//generate traj
t := count*deltaT;
landVel := -0.05 / period;
decTime := 0.1;
IF isContact(count,legID) = FALSE THEN
	IF t <= allContactTime + period THEN
		objSpline(x:=tp,y:=xp,dy0:=0,dy4:=0,      xt:=t,yt=>tipPos[legID].data[0],vt=>tipVel[legID].data[0]);
		objSpline(x:=tp,y:=yp,dy0:=0,dy4:=0,      xt:=t,yt=>tipPos[legID].data[1],vt=>tipVel[legID].data[1]);
		objSpline(x:=tp,y:=zp,dy0:=0,dy4:=landVel,xt:=t,yt=>tipPos[legID].data[2],vt=>tipVel[legID].data[2]);
	ELSE
		tipPos[legID].data[2] := tipPos[legID].data[2] + landVel*deltaT;//到达目标位置后继续下探
	END_IF
ELSE
	//强制停止，没有减速过程。减速过程的运动距离会导致机器人被顶起来
	FOR i:=0 TO 2 DO
		tipPos[legID].data[i] := tipPos[legID].data[i];
		tipVel[legID].data[i] := 0;
	END_FOR
	(*IF VecNorm(tipVel[legID]) > 1E-3 THEN
		FOR i:=0 TO 2 DO
			acc := -tipVel[legID].data[i] / decTime;
			tipPos[legID].data[i] := tipPos[legID].data[i] + tipVel[legID].data[i]*deltaT + 0.5*acc*deltaT*deltaT;
			tipVel[legID].data[i] := tipVel[legID].data[i] + acc*deltaT;
		END_FOR
	ELSE
		FOR i:=0 TO 2 DO
			tipPos[legID].data[i] := tipPos[legID].data[i];
			tipVel[legID].data[i] := 0;
		END_FOR
	END_IF*)
END_IF
END_METHOD

METHOD UpdateInitAndTrgt : BOOL
VAR_INPUT
END_VAR
VAR
	i: INT;
	bodyDist2T: Vec3;
	tipBias : Vec3;
	rotHalfYaw : Mat3;
END_VAR
//1.确定身体初始和目标位置、速度
//位置速度更新
bodyPosInit := bodyPos;
bodyVelInit := bodyVel;
bodyRPYInit := bodyRPY;
bodyOmgInit := bodyOmg;

//位姿计算：姿态在地面坐标系描述，位置在bodyTrgt坐标系描述
bodyRPYTrgt.data[2] := bodyRPYInit.data[2] + stepYaw;//yaw
CalcSlope(yaw := bodyRPYTrgt.data[2],
		  roll => bodyRPYTrgt.data[0], pitch => bodyRPYTrgt.data[1],
		  deltaH => bodyDist2T.data[2],tipDelta => tipBias);
//bodyRPYTrgt.data[0] := gvl.rpy_model[0] + bodyRPYTrgt.data[0] - bodyRPYInit.data[0];//引入实际角度修正
//bodyRPYTrgt.data[1] := gvl.rpy_model[1] + bodyRPYTrgt.data[1] - bodyRPYInit.data[1];//引入实际角度修正
objRotMtx(yaw:=bodyRPYTrgt.data[2],pitch:=bodyRPYTrgt.data[1],roll:=bodyRPYTrgt.data[0],
		  rm=>bodyPmxTrgt);

Arc2Line(arcLen:=stepL,angle:=stepYaw,lineLen=>stepL);
bodyDist2T.data[0] := stepL*COS(stepDir)*COS(-stepYaw/2)-stepL*SIN(stepDir)*SIN(-stepYaw/2);//身体转yaw时，位置只转yaw/2
bodyDist2T.data[1] := stepL*COS(stepDir)*SIN(-stepYaw/2)+stepL*SIN(stepDir)*COS(-stepYaw/2);

bodyPosTrgt := VecAdd(bodyPosInit,MatMulVec(bodyPmxTrgt,bodyDist2T));
bodyPosInit2T := VecNeg(bodyDist2T);
bodyVelInit2T := MatMulVec(MatTranspose(bodyPmxTrgt),bodyVelInit);

//2.确定摆动腿初始和目标位置，速度总为0
tipPosInit := tipPos;

objRotMtx(yaw:=stepYaw/2,pitch:=0,roll:=0,rm=>rotHalfYaw);
FOR i:=0 TO 5 DO
	tipPosTrgt2T[i] := MatMulVec(rotHalfYaw,VecAdd(tipPosTrgtBase[i],SetVec3(stepL/2*COS(stepDir),stepL/2*SIN(stepDir),0)));
	//tipPosTrgt[i] := VecAdd(VecAdd(MatMulVec(bodyPmxTrgt,tipPosTrgt2T[i]),bodyPosTrgt),tipBias);
	tipPosTrgt[i] := VecAdd(MatMulVec(bodyPmxTrgt,tipPosTrgt2T[i]),bodyPosTrgt);
END_FOR
END_METHOD

METHOD WatchDog : BOOL
VAR_INPUT
	count: UDINT;
END_VAR
IF isFeed=TRUE THEN
	starveCount := count + TRUNC(gvl.sampleRate*0.5);//0.5 second
	isFeed := FALSE;
END_IF

IF count>=starveCount THEN
	cmdL := 0;
	cmdLa := 0;
	cmdYaw := 0;
END_IF
END_METHOD

END_FUNCTION_BLOCK

// ---- POUs/tools/VectorMath/VecNormalize.TcPOU
FUNCTION VecNormalize : Vec3
VAR_INPUT
	a : Vec3;
END_VAR
VAR
END_VAR

VecNormalize := VecMulNum(a, 1/VecNorm(a));

END_FUNCTION

// ---- POUs/tools/VectorMath/VecNorm.TcPOU
FUNCTION VecNorm : lreal
VAR_INPUT
	a : Vec3;
END_VAR
VAR
END_VAR

VecNorm := SQRT(a.data[0] * a.data[0] + a.data[1] * a.data[1] + a.data[2] * a.data[2]);

END_FUNCTION

// ---- POUs/tools/VectorMath/VecCross.TcPOU
FUNCTION VecCross : Vec3
VAR_INPUT
	a, b : Vec3;
END_VAR
VAR
	a1, a2, a3 : LREAL;
	b1, b2, b3 : LREAL;
END_VAR

a1 := a.data[0];
a2 := a.data[1];
a3 := a.data[2];
b1 := b.data[0];
b2 := b.data[1];
b3 := b.data[2];

VecCross.data[0] := a2*b3 - a3*b2;
VecCross.data[1] := a3*b1 - a1*b3;
VecCross.data[2] := a1*b2 - a2*b1;

END_FUNCTION

// ---- POUs/tools/VectorMath/Atan2.TcPOU
FUNCTION Atan2 : LREAL//输出角度范围为[-pi,pi]
VAR_INPUT
	y : LREAL;
	x : LREAL;
END_VAR
VAR
END_VAR

IF ABS(x)<1E-6 THEN
	IF y>=0 THEN
		Atan2 := pi/2;
	ELSE
		Atan2 := -pi/2;
	END_IF
ELSE
	IF x<0 AND y>=0 THEN
		Atan2 := ATAN(y/x) + pi;
	ELSIF x<0 AND y<0 THEN
		Atan2 := ATAN(y/x) - pi;
	ELSE
		Atan2 := ATAN(y/x);
	END_IF
END_IF

END_FUNCTION

// ---- POUs/HardwareSetup/SdoSetup.TcPOU
FUNCTION_BLOCK SdoSetup
VAR_INPUT
END_VAR
VAR_OUTPUT
END_VAR
VAR
	bInitTrqSensorSDOCompleted        : ARRAY[0..2]  OF BOOL := [TRUE, FALSE, FALSE];
	bInitMotorDriveSDOCompleted       : ARRAY[0..18]  OF BOOL := [TRUE, FALSE, FALSE, FALSE, FALSE, FALSE, FALSE, 
                                                                  FALSE, FALSE, FALSE, FALSE, FALSE, FALSE,FALSE,FALSE,FALSE,FALSE,FALSE,FALSE];
	//trqSensorSdoSetup       : ARRAY[1..2]  OF TrqSensorSetup;
	driveSdoSetup           : ARRAY[1..18] OF MotorDriveSetup;
	trqSensorAdds           : ARRAY[1..3]  OF UINT := [1019, 1020,1021];
	driveAdds               : ARRAY[1..18] OF UINT := [1001, 1002, 1003,
                                                       1004, 1005, 1006,
                                                       1007, 1008, 1009,
                                                       1010, 1011, 1012,
                                                       1013, 1014, 1015,
                                                       1016, 1017, 1018];
													   
END_VAR

METHOD PUBLIC InitSdoConfig : BOOL
VAR_INPUT
END_VAR

VAR
	i: INT;
END_VAR
(*FOR i := 1 TO 2 DO
	IF bInitTrqSensorSDOCompleted[i-1] AND NOT bInitTrqSensorSDOCompleted[i] THEN // yk 第一个板子写完再写第二个，依次进行，0号值为true
		trqSensorSdoSetup[i].InitSDOs(board_id := i, bCompleted => bInitTrqSensorSDOCompleted[i]);
	END_IF
END_FOR

IF bInitTrqSensorSDOCompleted[1] AND bInitTrqSensorSDOCompleted[2] THEN
	FOR i := 1 TO 12 DO
		IF bInitMotorDriveSDOCompleted[i-1] AND NOT bInitMotorDriveSDOCompleted[i] THEN // 同理写完一个再写下一个，1ms刷新整个程序，for循环执行一次是微秒级，但是硬件写需要一定时间。
			driveSdoSetup[i].InitHomeConfig(bCompleted => bInitMotorDriveSDOCompleted[i]);
		END_IF
	END_FOR
END_IF
*)

	FOR i := 1 TO 18 DO//yk 如果调试1条腿，需要将其改为2
		IF bInitMotorDriveSDOCompleted[i-1] AND NOT bInitMotorDriveSDOCompleted[i] THEN // 同理写完一个再写下一个，1ms刷新整个程序，for循环执行一次是微秒级，但是硬件写需要一定时间。
			//driveSdoSetup[i].InitHomeConfig(bCompleted => bInitMotorDriveSDOCompleted[i]);
			driveSdoSetup[i].SetVelocityUnit(bCompleted => bInitMotorDriveSDOCompleted[i]);
		END_IF
	END_FOR
END_METHOD

METHOD PUBLIC SetSlaveAddr : BOOL//设置从站地址和home位置记为0,sdo相关编码从1到18
VAR_INPUT
END_VAR
VAR
	i : INT;
END_VAR
(*
FOR i := 1 TO 2 DO
	trqSensorSdoSetup[i].SetSlaveAddr(sNetId := '169.254.112.4.6.1', nSlaveAddr := trqSensorAdds[i]);
END_FOR
*)

FOR i := 1 TO 18 DO     //yk 写1号到18号驱动器的home参数
	//driveSdoSetup[i].SetSlaveAddr(sNetId := '120.1.1.15.4.1', nSlaveAddr := driveAdds[i]);//冰壶1参数
	driveSdoSetup[i].SetSlaveAddr(sNetId := '10.0.0.119.4.1', nSlaveAddr := driveAdds[i]);//冰壶2参数
	//driveSdoSetup[i].SetHomeOffset(LREAL_TO_DINT(gvl.posHomeOffsets[i-1]/180.0*pi/gvl.count2radianRatio));
	//driveSdoSetup[i].SetHomeOffset(0);
END_FOR
END_METHOD

END_FUNCTION_BLOCK

// ---- POUs/HardwareSetup/MotorDriveSetup.TcPOU
FUNCTION_BLOCK MotorDriveSetup
VAR_INPUT
END_VAR
VAR_OUTPUT
END_VAR
VAR
	// hardware address
    netId		: T_AmsNetId := '120.1.1.15.4.1'; (* NetId of EtherCAT Master *)
    slaveAddr	: UINT       := 1001; (* Port Number of EtherCAT Slave *)
	//homeOffset  : DINT       := 0;
	//homeMethod  : BYTE       := 35;
	//isCompleted : ARRAY[0..1] OF BOOL := [FALSE, FALSE];
	isCompleted:BOOL:=FALSE;
	//VelocityOptions: UDINT:=16#FDB44700;
	VelocityOptions: UDINT:=16#FEB44700; 
	//isAllCompleted : BOOL := FALSE;
END_VAR

METHOD PUBLIC InitHomeConfig : BOOL
VAR_INPUT
END_VAR
VAR_OUTPUT
	bCompleted : BOOL := FALSE;
END_VAR
VAR
	nIndexAdd : WORD := 16#607C;
	i : BYTE;
END_VAR
(*IF NOT isCompleted[0] THEN
	gvl.sdoWriteOnce(sNetId := netId, nSlaveAddr := slaveAddr,
					 nIndex := 16#607C, nSubIndex := 0, pSrcBuf := ADR(homeOffset), 
					 cbBufLen := SIZEOF(DINT), bComplAcc := FALSE, bWriteOnce=> isCompleted[0]);
END_IF

IF isCompleted[0] AND NOT isCompleted[1] THEN
	gvl.sdoWriteOnce(sNetId := netId, nSlaveAddr := slaveAddr,
					 nIndex := 16#6098, nSubIndex := 0, pSrcBuf := ADR(homeMethod), 
					 cbBufLen := SIZEOF(DINT), bComplAcc := FALSE, bWriteOnce=> isCompleted[1]);
END_IF

isAllCompleted := isCompleted[0] AND isCompleted[1];
bCompleted := isAllCompleted;*)
END_METHOD

METHOD PUBLIC SetHomeOffset : BOOL
VAR_INPUT
	hmOffset : DINT;
END_VAR
//homeOffset := hmOffset;
END_METHOD

METHOD PUBLIC SetSlaveAddr : BOOL
VAR_INPUT
	sNetId		: T_AmsNetId;
    nSlaveAddr	: UINT ;
END_VAR
VAR

END_VAR
netId	    := sNetId; 
slaveAddr	:= nSlaveAddr;
END_METHOD

METHOD PUBLIC SetVelocityUnit : BOOL
VAR_INPUT
END_VAR
VAR_OUTPUT
	bCompleted : BOOL := FALSE;
END_VAR
VAR
	nIndexAdd : WORD := 16#60A9;
	i : BYTE;
END_VAR
IF NOT isCompleted THEN
	gvl.sdoWriteOnce(sNetId := netId, nSlaveAddr := slaveAddr,
					 nIndex := 16#60A9, nSubIndex := 0, pSrcBuf := ADR(VelocityOptions), 
					 cbBufLen := SIZEOF(UDINT), bComplAcc := FALSE, bWriteOnce=> isCompleted);
END_IF
bCompleted := isCompleted;
END_METHOD

END_FUNCTION_BLOCK

// ---- POUs/controller/IntegratedDrive.TcPOU
FUNCTION_BLOCK PUBLIC IntegratedDrive//和驱动器有关数组都按照每条腿的小腿、大腿、侧摆顺序给定,编码0-17
VAR_INPUT
END_VAR
VAR_OUTPUT
END_VAR
VAR
	motor              : Motor;
	//motor_targetVel:dint;
	motor_targetVel:lreal;
	trqSensor          : TorqueSensor;
	
	statusMode         : UINT;
	statusDispStr      : STRING(25);
	opModeDispStr      : STRING(25);
	enableBit          : BOOL;
	setAck             : UINT;
	isHomeSwitchOn     : BOOL;
	
	reductionRatio     : LREAL := 50.0;
    positionHomeOffset : LREAL;
	positionOffset     : LREAL := -1.3781499114412897226085228010063;
	count2radianRatio  : LREAL := 2*pi/1048576;  // 2*pi/1048576
	motorAngle         : LREAL;// 电机实际角度值
	motorAngVel        : LREAL;
	motorDir           : INT   := 1;
	
	tgtAngle           : LREAL := 4.71238898; // 1.5 * pi  yk 电机目标角度值
	tgtAngVel          : LREAL := 0;
	addTorque          : LREAL := 0;
	
	isHomeSetMode      : BOOL;
	inHomeModeCount    : UINT;
	isHoming           : BOOL;
	//homeVel            : dint := 2000;// 2000 inc/s
	homeVel            : LREAL := 0.01;// 0.1rad/s
	
	cvSetVel           : LREAL := 0;
	cvStart            : BOOL;
	cvStop             : BOOL;
	cvCount            : DINT := 0;
	
	trqSensorDir       : INT   := 1;
	trqFiltered        : LREAL := 0;
	trqDotFiltered     : LREAL := 0;
	trqCalibrated      : LREAL := 0;
	
	isInForceControl   : BOOL := FALSE;
	forceModeCount     : UDINT := 0;
	trqErrSumLast      : LREAL := 0;
	trqOutput          : LREAL := 0;
	
	kVirtual           : LREAL := 220; //SQ
	bVirtual           : LREAL := 25;//SQ
	//kVirtual           : LREAL := 0;
	//bVirtual           : LREAL := 0;
	//reducerColbConstant: LREAL := 0.0 * 100;
	reducerColbConstant: LREAL := 0.01 * 100;
	
	kpTrqLoop          : LREAL := 0.5; 
	kiTrqLoop          : LREAL := 0.75;
	trqCmdLimit        : LREAL := 130;
	
	trqControlAngRange : ARRAY[0..1] OF LREAL := [3.51, 5.91];
	trqConstant        : LREAL := 0.11;
	curMax             : LREAL := 13;
	
	faultCount         : UINT  := 0;
	
	motorActualPosLimit:DINT:=0;
	motorActualPosUpperLimit:DINT:=524288;
	motorActualPosLowerLimit:DINT:=-524288;
	motorStepIncrement:DINT:=1048576;
	//velocityUnitRatio:LREAL:=0.001;//0.001rpm
	velocityUnitRatio:LREAL:=0.01;//0.01rpm
	
	index:UINT:=0;//motor sequence number
	motorActualHomePosIncrement:DINT:=0;
	
	//absMove
	IsAbsMoveState:BOOL:=FALSE;
	cpStart:BOOL:=FALSE;
	cpStop:BOOL:=FALSE;
	AbsMoveTgtPos:LREAL;
	cpCount            : DINT := 0;
	cpStartAngle:LREAL;
	cpRefAngle:LREAL;
	
END_VAR

METHOD PUBLIC AbsMove : BOOL
VAR_INPUT
END_VAR

VAR CONSTANT
	ACC_TOTAL_CNT:   DINT := 2000;
END_VAR
IF index=18 OR index=19 OR index=20 THEN
		count2radianRatio:=2*pi/4096.0/9.0;
ELSE
		count2radianRatio:=2*pi/1048576.0;	
END_IF

IF cpStart=TRUE THEN
	IF cpCount < ACC_TOTAL_CNT THEN
		cpRefAngle:=cpStartAngle+(AbsMoveTgtPos-cpStartAngle)* SIN(0.5 * pi * cvCount / ACC_TOTAL_CNT);
	  	cpCount := cpCount + 1; 
   	ELSE
	  cpRefAngle := AbsMoveTgtPos;
   	END_IF 
	motor.targetPos:= motorDir*TRUNC((cpRefAngle-positionHomeOffset+positionOffset)/count2radianRatio);
ELSE
	motor.targetPos:=motor.actualPos;
END_IF
IF cpStop=TRUE THEN
	motor.targetPos:=motor.actualPos;
	cpStart:=FALSE;
	IsAbsMoveState:=FALSE;
	cpCount:=0;
END_IF
END_METHOD

METHOD PUBLIC CalculateCurrentCmd : BOOL
VAR_INPUT
END_VAR
VAR
	curCmd: DINT;
END_VAR
curCmd := TRUNC(trqOutput / reductionRatio / trqConstant / curMax * 1000); //yk 扭矩常数和最大电流进行折算，还有一种通过，扭矩常数和最大电流乘积就是最大扭矩
motor.targetTrq := motorDir * DINT_TO_INT(curCmd);
END_METHOD

METHOD PUBLIC CalculateMotorAngle : INT
VAR_INPUT
END_VAR
//motorAngVel := motorDir * motor.actualVel * count2radianRatio;
IF index=18 OR index=19 or index=20 THEN
	motorAngVel := motorDir * motor.actualVel *2.0*pi/(9.0*4096.0);
ELSE
	motorAngVel := velocityUnitRatio*motorDir * motor.actualVel *2*pi/60/ 50;//rpm motor.actualVel在电机上折算,正确
END_IF

//motorAngVel := velocityUnitRatio*motorDir * motor.actualVel *2*pi/60;//rpm motor.actualVel在腿上折算

motorActualPosLimit:=motor.actualPos;
motorActualPosLimit:=TRUNC(AngleCutFun(angRow:=motorActualPosLimit , upper:=motorActualPosUpperLimit , lower:=motorActualPosLowerLimit , rangLength:=motorStepIncrement ));

motorActualHomePosIncrement:=TRUNC(AngleCutFun(angRow:=motorActualHomePosIncrement , upper:=motorActualPosUpperLimit , lower:=motorActualPosLowerLimit , rangLength:=motorStepIncrement ));
IF index<>20 THEN
	//positionOffset:=motorActualHomePosIncrement;
	positionOffset := motorDir * motorActualHomePosIncrement * count2radianRatio;
END_IF

motorAngle := motorDir * motorActualPosLimit * count2radianRatio - positionOffset + positionHomeOffset;// yk positionOffset是home位置对应编码器数值，positionHomeOffset是找home停止位置对应的弧度,老的编程方式需要记录当前home处count值给positionoffset，新的编程其值为0

IF  index=2 OR index=3 OR index=5 OR index=6 OR index=8 OR index=9 OR index=11 OR index=12 OR index=14 OR index=17 THEN
	motorAngle:=AngleCutFun(angRow:=motorAngle , upper:=pi , lower:=-pi , rangLength:=2*pi );
END_IF

IF index=1 OR index=4 OR index=7 OR index=10 OR index=13 OR index=16 OR index=0 OR  index=15 THEN
	motorAngle:=AngleCutFun(angRow:=motorAngle , upper:=2*pi , lower:=0 , rangLength:=2*pi );
END_IF


CalculateMotorAngle := 0;
END_METHOD

METHOD PUBLIC CalibrateTrqData : BOOL
VAR_INPUT
END_VAR
VAR_STAT
END_VAR
VAR
	LPFilter : LowpassFilter;
	trqSensorRawData      : LREAL;
END_VAR
trqSensorRawData := trqSensor.trqsensorValue;

IF trqSensorRawData > 0 THEN
	trqSensorRawData := trqSensorRawData / trqSensor.signalPosSlope;
ELSE
	trqSensorRawData := trqSensorRawData / trqSensor.signalNegSlope;
END_IF

trqSensorRawData := trqSensorDir * trqSensorRawData;

LPFilter(x := trqSensorRawData,
	     y := trqFiltered,
		 ydot := trqDotFiltered,
		 yout => trqFiltered,
		 ydotout => trqDotFiltered);

trqCalibrated := trqFiltered;
//trqCalibrated := trqSensorRawData;
END_METHOD

METHOD PUBLIC DriverControl : BOOL
VAR_INPUT
	operationModeCmd : USINT;
	enableCmd        : BOOL;
END_VAR
motor.opMode := operationModeCmd;

///////////////////////////////////////////////////////////////////////////////////////yk???????
IF isHomeSetMode THEN
	motor.opMode := 6;
	IF motor.opModeDisp = 6 THEN
		inHomeModeCount := inHomeModeCount + 1;
	END_IF
END_IF

IF enableCmd = TRUE AND enableBit = FALSE THEN     	 (*Enable driver*)
	CASE statusMode OF
		(*0,32:;*)                               (*NOT READY TO SWITCH ON*)
		64,96:  motor.ctrlWord := 6;             (*SWITCH ON DISABLED*)
		33:     motor.ctrlWord := 7;             (*READY TO SWITCH ON*)
		35:     motor.ctrlWord := 15;            (*SWITCHED ON*)
		39:;                                     (*OPERATION ENABLED*)
		7:      motor.ctrlWord := 15;            (*QUICK STOP ACTIVE*)
		4:      motor.ctrlWord := 15;
		(*15,47:controlword:=128;                (*FAULT REACTION ACTIVE*)
		8,40:controlword:=128;*)                 (*FAULT*)
		ELSE    motor.ctrlWord := 128; 
	END_CASE
	//trqErrSumLast := 0;
ELSIF enableCmd = FALSE AND enableBit = TRUE  THEN
	motor.ctrlWord := 0;                         (*Disable driver*)	
END_IF 

IF isHomeSetMode THEN
	IF statusMode = 39 AND motor.opModeDisp = 6 AND inHomeModeCount > 20 THEN
		IF setAck = 0 THEN
			motor.ctrlWord := 31;//yk 31=2# 1_1111,home开始
		ELSE
			motor.ctrlWord := 15;
			isHomeSetMode := FALSE;
		END_IF
	END_IF
END_IF

motor.maxTrq := 2500;
DriverControl := TRUE;
END_METHOD

METHOD PUBLIC GoHome : BOOL
VAR_INPUT
END_VAR
// Handle homing state
IF isHoming THEN
	IF isHomeSwitchOn THEN
		cvStop := TRUE;
		cvStart := FALSE;
		isHoming := FALSE;
	END_IF
END_IF
END_METHOD

METHOD PUBLIC ImpedControl : BOOL
VAR_INPUT
    desiredTorque : LREAL;
	isExternalIC  : BOOL;
END_VAR
VAR_OUTPUT
	curCmd: DINT;
END_VAR
VAR
	measuredTrq : LREAL;
	posError : LREAL;
	velError : LREAL;
	trqCmd: LREAL;
	
	coulombFric: LREAL;
	signOfVel: LREAL;
	trqErr: LREAL;
	trqCorrection: LREAL;

	trqCmd2: LREAL;

	minDistanceMotor: LREAL;
END_VAR
measuredTrq := trqCalibrated;
posError := motorAngle - tgtAngle;
IF ABS(posError)>pi THEN
	minDistanceMotor:=MinDistanceValue(motorAngle,tgtAngle);
	posError :=minDistanceMotor - tgtAngle;
END_IF
velError := motorAngVel - tgtAngVel;

IF isExternalIC THEN
	trqCmd := desiredTorque;
ELSE
	trqCmd := -kVirtual * posError - bVirtual * velError + addTorque;  // Impedance control
END_IF
//trqCmd := 0;   // Following control

// deadzone for torque measurement
IF ABS(measuredTrq) < 0.15 THEN
	measuredTrq := 0;
END_IF

signOfVel := 0;
IF motorAngVel > 0.001 THEN
	signOfVel := 1;
END_IF
IF motorAngVel < -0.001 THEN
	signOfVel := -1;
END_IF

coulombFric := signOfVel * reducerColbConstant;

//////////////////////////////////////////////////////////////////////////////////////////
//扭矩传感器数据用来搭电流环
trqErr := trqCmd - (-measuredTrq);//yk 扭矩方向和标定方向正负关系决定
//trqErr := trqCmd - (measuredTrq);//yk 扭矩方向和标定方向正负关系决定
trqErrSumLast := trqErrSumLast + trqErr / DINT_TO_LREAL(gvl.sampleRate);
trqCorrection := kpTrqLoop * trqErr + kiTrqLoop * trqErrSumLast;

trqCmd2 := trqCmd + coulombFric + trqCorrection;

IF trqCmd2 > trqCmdLimit THEN
	trqCmd2 := trqCmdLimit;
END_IF
IF trqCmd2 < -trqCmdLimit THEN
	trqCmd2 := -trqCmdLimit;
END_IF
//////////////////////////////////////////////////////////////////////////////////////////

(*IF motorAngle < trqControlAngRange[0] THEN
	trqCmd2 := 0;
	trqErrSumLast := 0;
END_IF
IF motorAngle > trqControlAngRange[1] THEN
	trqCmd2 := 0;
	trqErrSumLast := 0;
END_IF*)

trqOutput := trqCmd2;

ImpedControl := TRUE;
END_METHOD

METHOD PUBLIC InitParam : BOOL
VAR_INPUT
	motorDirIn     : INT;
	trqSensorDirIn : INT;
	posHomeOffsetIn: LREAL;

	signalPosSlope : LREAL;
	signalNegSlope : LREAL;
	redcClbConst   : LREAL;
	
	//homingVel      : DINT;
	homingVel      : lreal;
	trqCtrlUpperAng: LREAL;
	trqCtrlLowerAng: LREAL;
	tgtAngleIn  : LREAL;
	motorActualHomePosIncrementIn:DINT;
	indexIn:UINT;
	
	kVirtualIn:LREAL;
	bVirtualIn:LREAL;
	kpTrqLoopIn:LREAL;
	kiTrqLoopIn:LREAL;
	count2radianRatioIn:LREAL;
	
END_VAR
motorDir           := motorDirIn;
THIS^.trqSensorDir := trqSensorDirIn;
positionHomeOffset := posHomeOffsetIn;

trqSensor.signalNegSlope := signalNegSlope;
trqSensor.signalPosSlope := signalPosSlope;

homeVel             := homingVel;
reducerColbConstant := redcClbConst;

trqControlAngRange[1] := trqCtrlUpperAng;
trqControlAngRange[0] := trqCtrlLowerAng;
tgtAngle              := tgtAngleIn;
tgtAngVel             := 0;
addTorque             := 0;
motorActualHomePosIncrement:=motorActualHomePosIncrementIn;
index:=indexIn;
kVirtual:=kVirtualIn;
bVirtual:=bVirtualIn;
kpTrqLoop:=kpTrqLoopIn;
kiTrqLoop:=kiTrqLoopIn;
count2radianRatio:=count2radianRatioIn;



InitParam := TRUE;
END_METHOD

METHOD JogControl : BOOL
VAR_INPUT
END_VAR

VAR CONSTANT
	ACC_TOTAL_CNT:   DINT := 500;
END_VAR
IF cvStart THEN
   IF cvCount < ACC_TOTAL_CNT THEN
	  motor_targetVel := motorDir * TRUNC(cvSetVel * SIN(0.5 * pi * cvCount / ACC_TOTAL_CNT)); 
	  cvCount := cvCount + 1; 
   ELSE
	  motor_targetVel := motorDir * cvSetVel;
   END_IF   
END_IF

IF cvStop THEN
   cvStart:=FALSE;   
   IF cvCount > 0 THEN
	  motor_targetVel := motorDir * TRUNC(cvSetVel * SIN(0.5 * pi * cvCount / ACC_TOTAL_CNT)); 
	  cvCount := cvCount - 1; 
   ELSE
	  cvCount := 0;	  
	  motor_targetVel := motorDir * 0;
      cvStop:=FALSE;
   END_IF
END_IF

//motor.targetVel:= TRUNC(1/velocityUnitRatio*motor_targetVel*60/(2*pi));//腿端
IF index=18 OR index=19 OR index=20 THEN
	motor.targetVel:=TRUNC(motor_targetVel*9.0/(2*pi)*4096);
ELSE
	motor.targetVel:= TRUNC(1.0/velocityUnitRatio*motor_targetVel*60.0/(2*pi)*50.0);//电机端,确认
END_IF
END_METHOD

METHOD PUBLIC SetImpdTarget : BOOL
VAR_INPUT
	//yk  按照小腿、大腿、侧摆顺序给出;不是按照单腿运动学中侧摆角、大腿角、小腿角给出（小腿角加了pi）,在DownloadDriveCmds 中折算
	targetPos, targetVel, additionalFce : LREAL;
END_VAR
tgtAngle := targetPos;
tgtAngVel := targetVel;
addTorque := additionalFce;
END_METHOD

METHOD PUBLIC SetImpedanceParam : BOOL
VAR_INPUT
	kp, kd, kptrq, kitrq : LREAL;
END_VAR
kVirtual := kp;
bVirtual := kd;
kpTrqLoop  := kptrq;
kiTrqLoop  := kitrq;
END_METHOD

METHOD PUBLIC SetInitPosition : BOOL
VAR_INPUT
END_VAR

motorActualPosLimit:=motor.actualPos;
WHILE(motorActualPosLimit>motorActualPosUpperLimit OR motorActualPosLimit<motorActualPosLowerLimit) DO
	IF motorActualPosLimit>motorActualPosUpperLimit THEN
		motorActualPosLimit:=motorActualPosLimit-motorStepIncrement;
	ELSE
		motorActualPosLimit:=motorActualPosLimit+motorStepIncrement;			
	END_IF
END_WHILE

positionOffset := motorDir * motorActualPosLimit * count2radianRatio;

//isHomeSetMode      := TRUE;
isHomeSetMode      := false;
inHomeModeCount    := 0;
SetInitPosition    := FALSE;
END_METHOD

METHOD PUBLIC SetTrgVel : BOOL
VAR_INPUT
	trgVelIn:lreal;
END_VAR
cvSetVel:=trgVelIn;
motor.targetVel:=motorDir *TRUNC(trgVelIn*9.0/(2*pi)*4096);
motor_targetVel := motorDir * cvSetVel;
END_METHOD

METHOD PUBLIC StartAbsMove : BOOL
VAR_INPUT
	AbsMoveTgtPosIn:lreal;
END_VAR
IsAbsMoveState:=TRUE;
AbsMoveTgtPos:=AbsMoveTgtPosIn;
cpStart:=TRUE;
cpStop:=FALSE;
cpStartAngle:=motorAngle;
cpCount :=0;
END_METHOD

METHOD PUBLIC StartForceControl : BOOL
VAR_INPUT
END_VAR
// check force ctrl condition
IF NOT enablebit THEN
	StartForceControl := FALSE;
	RETURN;
END_IF

// change control mode flag
isInForceControl := TRUE;


// set normal angle and angvel
tgtAngle := motorAngle;
tgtAngVel := 0;
addTorque := 0;

// reset force control integration
trqErrSumLast := 0;

// set force control count
forceModeCount := 1;

StartForceControl := TRUE;
END_METHOD

METHOD PUBLIC StartGoHome : BOOL
VAR_INPUT
END_VAR
isHoming := TRUE;
cvSetVel := homeVel;
cvStart  := TRUE;
cvStop   := FALSE;
END_METHOD

METHOD PUBLIC StartJog : BOOL
VAR_INPUT
	//jogVelocity : DINT;
	jogVelocity :lreal;
END_VAR
cvSetVel := jogVelocity;
cvStart  := TRUE;
cvStop   := FALSE;
END_METHOD

METHOD PUBLIC StatusDisplay : BOOL
VAR_INPUT
END_VAR
statusMode := motor.statusWord AND 2#0000_0000_0110_1111;//取出6个1对应的位
setAck:= motor.statusWord AND 2#0001_0000_0000_0000;  //yk home模式下1代表找home出错，0代表home过程中没有错,找home时使用
isHomeSwitchOn := (DINT_TO_UDINT(motor.digInputs) AND 2#0001_0000_0000_0000_0000_0000) = 2#0001_0000_0000_0000_0000_0000;//yk 17到21位为数字输入信号,home开关在第5个input口，所以第21位取出来，驱动器tuning时可以找到第几个输入,对应即可

(* Axis status display *)
CASE statusMode OF
	(*0,32:;*)                                  (*NOT READY TO SWITCH ON*)
	64,96 : statusDispStr := 'DISABLED';        (*SWITCH ON DISABLED*)//2#100_0000,2#110_0000,
	33    : statusDispStr := 'READY TO POWON';  (*READY TO SWITCH ON*)//2#010_0001
	35    : statusDispStr := 'POWERED ON';      (*SWITCHED ON*)//2#010_0011
	39    : statusDispStr := 'ENABLED';         (*OPERATION ENABLED*)//2#010_0111
	7     : statusDispStr := 'QUICK STOP';      (*QUICK STOP ACTIVE*)//2#000_0111
	(*15,47:controlword:=128;                   (*FAULT REACTION ACTIVE*)
	8,40:controlword:=128;*)                    (*FAULT*)
	ELSE statusDispStr:='FAULT';
END_CASE
(* set enable bit *)
IF statusMode = 39 THEN
	enableBit := TRUE;
ELSE
	enableBit := FALSE;
END_IF

IF statusDispStr = 'FAULT' THEN
	faultCount := faultCount + 1;
ELSE
	faultCount := 0;
END_IF

(*IF faultCount > 1 THEN
	gvl.emergencyStop := TRUE;
END_IF*)

CASE motor.opModeDisp OF
    -1: opModeDispStr  := 'No mode';
	0 : opModeDispStr  := 'Reserved';
	1 : opModeDispStr  := 'Profiled pos';
	2 : opModeDispStr  := 'Velocity';
	3 : opModeDispStr  := 'Profile vel';
	4 : opModeDispStr  := 'Profiled trq';
	5 : opModeDispStr  := 'Reserved';
	6 : opModeDispStr  := 'Homing mode';
	7 : opModeDispStr  := 'Inter position';
	8 : opModeDispStr  := 'Syn pos cycle';
	9 : opModeDispStr  := 'Syn vel cycle';
	10: opModeDispStr  := 'Syn trq cycle';
	ELSE 
        opModeDispStr  := 'Reserved';
END_CASE

StatusDisplay := TRUE;
END_METHOD

METHOD PUBLIC StopAbsMove : BOOL
VAR_INPUT
END_VAR
IsAbsMoveState:=FALSE;
cpStart:=FALSE;
cpStop:=TRUE;
cpCount :=0;
END_METHOD

METHOD PUBLIC StopForceControl : BOOL
VAR_INPUT
END_VAR
StopForceControl := TRUE;
// change control mode flag
isInForceControl := FALSE;

// set normal angle and angvel
tgtAngle  := motorAngle;
tgtAngVel := 0;
addTorque := 0;

motor.targetVel := 0;
motor.targetPos := motor.actualPos;
motor.targetTrq := 0;

// reset force control integration
trqErrSumLast := 0;

// reset force control count
forceModeCount := 0;
END_METHOD

METHOD PUBLIC StopJog : BOOL
VAR_INPUT
END_VAR
cvStart  := FALSE;
cvStop   := TRUE;
isHoming := FALSE;
END_METHOD

END_FUNCTION_BLOCK

// ---- POUs/tools/AngleCutFun.TcPOU
FUNCTION AngleCutFun : lreal
VAR_INPUT
	angRow:LREAL;
	upper:LREAL;
	lower:LREAL;
	rangLength:LREAL;
END_VAR
VAR
	angCutted:LREAL;
END_VAR

angCutted:=angRow;
WHILE(angCutted>upper OR angCutted<lower) DO
    IF angCutted>upper THEN
        angCutted:=angCutted-rangLength;
    else
        angCutted:=angCutted+rangLength;
    END_IF
END_WHILE
AngleCutFun:=angCutted;

END_FUNCTION

// ---- POUs/tools/LowpassFilter.TcPOU
FUNCTION_BLOCK LowpassFilter
VAR_INPUT
	x : LREAL;
	y : LREAL;
	ydot : LREAL;
END_VAR
VAR_OUTPUT
	yout : LREAL;
	ydotout : LREAL;
END_VAR
VAR
	cutFreq : LREAL := 100.0;
	wcut: LREAL := 2 * pi * cutFreq;
	w: LREAL := 1/wcut;
	wwcut : LREAL := 1/w/w;
	dt_: LREAL:= 1.0/DINT_TO_LREAL(gvl.sampleRate);
	yddot: LREAL;
END_VAR

yddot := wwcut*(x - y - 2 * 0.707 * w * ydot);
ydotout := ydot + yddot * dt_;
yout := y + ydotout * dt_;

END_FUNCTION_BLOCK

// ---- POUs/tools/SdoWrite.TcPOU
FUNCTION_BLOCK SdoWrite
VAR_INPUT
	sNetId      : T_AmsNetID;
	nSlaveAddr  : UINT;
	nIndex		: WORD; (* CoE Object Index *)
	nSubIndex	: BYTE; (* Subindex of CoE Object *)
	pSrcBuf		: PVOID; (* variable address to be written to the CoE Object *)
	cbBufLen	: UDINT; (* size of variable to be written *)
	bComplAcc	: BOOL;
END_VAR
VAR
	fbSdoWrite	: FB_EcCoESdoWriteEx;
    bError     : BOOL;
    nErrId     : UDINT;
END_VAR
VAR_OUTPUT
	bWriteOnce : BOOL := FALSE;
END_VAR

bWriteOnce := FALSE;
fbSdoWrite(
    sNetId     := sNetId,
    nSlaveAddr := nSlaveAddr,
    nIndex     := nIndex,
    nSubIndex  := nSubIndex,
    pSrcBuf    := pSrcBuf,
    cbBufLen   := cbBufLen,
	bCompleteAccess := bComplAcc,
    bExecute   := TRUE
);
IF NOT fbSdoWrite.bBusy THEN
  	IF NOT fbSdoWrite.bError THEN 
       	(* write successful *)
   		bError := FALSE;
   		nErrId := 0;
		bWriteOnce := TRUE;
    ELSE 
       	(* write failed *)
       	bError := fbSdoWrite.bError;
       	nErrId := fbSdoWrite.nErrId;
    END_IF
	fbSdoWrite(bExecute := FALSE);
END_IF

END_FUNCTION_BLOCK

// ---- POUs/controller/LegController.TcPOU
FUNCTION_BLOCK LegController
VAR_INPUT
END_VAR
VAR_OUTPUT
END_VAR
VAR 
	legId            : UINT;
	shankLength      : LREAL := 0.5;
	thighLength      : LREAL := 0.5;
	sagPlaneOffset	  :LREAL:=0.1246;
	
	motorAnglesIn    : ARRAY[0..2] OF LREAL := [0, 0, 0];//电机角度+0,0,pi,正运动学运算输入
	motorAngVelIn    : ARRAY[0..2] OF LREAL := [0, 0, 0];
	jointTorqueIn    : ARRAY[0..2] OF LREAL := [0, 0, 0];
	
	motorRefAnglesIn : ARRAY[0..2] OF LREAL := [0, 0, 0];
	
	motorAnglesOut   : ARRAY[0..2] OF LREAL := [0, 0, 0];
	motorAngVelOut   : ARRAY[0..2] OF LREAL := [0, 0, 0];
	jointTorqueOut   : ARRAY[0..2] OF LREAL := [0, 0, 0];

	phy2absMapping   : ARRAY[0..2] OF INT   := [2, 1, 0];
	//axisAngleOffset  : ARRAY[0..2] OF LREAL := [0, 0, pi];
	axisAngleOffset  : ARRAY[0..2] OF LREAL := [0, 0, 0];
END_VAR

METHOD PUBLIC DesireDriveForce : BOOL
VAR_INPUT
	fTipDes : ARRAY[0..2] OF LREAL;
	motorAng: ARRAY[0..2] OF LREAL;
	legIndex:INT;
END_VAR
VAR_OUTPUT
	fDrvDes : ARRAY[0..2] OF LREAL;
END_VAR
VAR
	thighAng : LREAL;
	shankAng : LREAL;
	xFTipdes : LREAL;
	yFTipdes : LREAL;
	zFTipDes: LREAL;
	abdctAng: LREAL;
	ySag: LREAL;
END_VAR
(*xFTipDes := fTipDes[0];
yFTipDes := fTipDes[1];
zFTipDes := fTipDes[2];

abdctAng := motorAng[0];
thighAng := motorAng[1];
shankAng := motorAng[2];

ySag := thighLength*SIN(thighAng) + shankLength*SIN(shankAng);

fDrvDes[0] := (-SIN(abdctAng)*ySag+cos(abdctAng)*sagPlaneOffset)*yFTipDes + (COS(abdctAng)*ySag+sin(abdctAng)*sagPlaneOffset)*zFTipDes;
fDrvDes[1] := -thighLength*SIN(thighAng)*xFTipDes + COS(abdctAng)*thighLength*COS(thighAng)*yFTipDes + SIN(abdctAng)*thighLength*COS(thighAng)*zFTipDes;
fDrvDes[2] := -shankLength*SIN(shankAng)*xFTipDes + COS(abdctAng)*shankLength*COS(shankAng)*yFTipDes + SIN(abdctAng)*shankLength*COS(shankAng)*zFTipDes;*)
IF legIndex=0 OR legIndex=5 THEN
	gvl.legCtrl[legIndex].DesireDriveForce_1(fTipDes:=fTipDes , motorAng:=motorAng , fDrvDes=> fDrvDes);
ELSE
	gvl.legCtrl[legIndex].DesireDriveForce_2(fTipDes:=fTipDes , motorAng:=motorAng , fDrvDes=> fDrvDes);
END_IF

DesireDriveForce := TRUE;
END_METHOD

METHOD PUBLIC DesireDriveForce_1 : BOOL
VAR_INPUT
	fTipDes : ARRAY[0..2] OF LREAL;
	motorAng: ARRAY[0..2] OF LREAL;
END_VAR
VAR_OUTPUT
	fDrvDes : ARRAY[0..2] OF LREAL;
END_VAR
VAR
	thighAng : LREAL;
	shankAng : LREAL;
	xFTipdes : LREAL;
	yFTipdes : LREAL;
	zFTipDes: LREAL;
	abdctAng: LREAL;
	ySag: LREAL;
END_VAR
xFTipDes := fTipDes[0];
yFTipDes := fTipDes[1];
zFTipDes := fTipDes[2];

abdctAng := motorAng[0];
thighAng := motorAng[1];
shankAng := motorAng[2];

ySag := thighLength*SIN(thighAng) + shankLength*SIN(shankAng);

fDrvDes[0] := (-SIN(abdctAng)*ySag+cos(abdctAng)*sagPlaneOffset)*yFTipDes + (COS(abdctAng)*ySag+sin(abdctAng)*sagPlaneOffset)*zFTipDes;
fDrvDes[1] := -thighLength*SIN(thighAng)*xFTipDes + COS(abdctAng)*thighLength*COS(thighAng)*yFTipDes + SIN(abdctAng)*thighLength*COS(thighAng)*zFTipDes;
fDrvDes[2] := -shankLength*SIN(shankAng)*xFTipDes + COS(abdctAng)*shankLength*COS(shankAng)*yFTipDes + SIN(abdctAng)*shankLength*COS(shankAng)*zFTipDes;

DesireDriveForce_1 := TRUE;
END_METHOD

METHOD PUBLIC DesireDriveForce_2 : BOOL
VAR_INPUT
	fTipDes : ARRAY[0..2] OF LREAL;
	motorAng: ARRAY[0..2] OF LREAL;
END_VAR
VAR_OUTPUT
	fDrvDes : ARRAY[0..2] OF LREAL;
END_VAR
VAR
	thighAng : LREAL;
	shankAng : LREAL;
	xFTipdes : LREAL;
	yFTipdes : LREAL;
	zFTipDes: LREAL;
	abdctAng: LREAL;
	ySag: LREAL;
END_VAR
xFTipDes := fTipDes[0];
yFTipDes := fTipDes[1];
zFTipDes := fTipDes[2];

abdctAng := motorAng[0];
thighAng := motorAng[1];
shankAng := motorAng[2];

ySag := thighLength*SIN(thighAng) + shankLength*SIN(shankAng+thighAng);

fDrvDes[0] := (-SIN(abdctAng)*ySag+cos(abdctAng)*sagPlaneOffset)*yFTipDes + (COS(abdctAng)*ySag+sin(abdctAng)*sagPlaneOffset)*zFTipDes;
fDrvDes[1] := -(thighLength*SIN(thighAng)+shankLength*SIN(shankAng+thighAng))*xFTipDes + COS(abdctAng)*(thighLength*COS(thighAng)+shankLength*COS(shankAng+thighAng))*yFTipDes + SIN(abdctAng)*(thighLength*COS(thighAng)+shankLength*COS(shankAng+thighAng))*zFTipDes;
fDrvDes[2] := -shankLength*SIN(shankAng+thighAng)*xFTipDes + COS(abdctAng)*shankLength*COS(shankAng+thighAng)*yFTipDes + SIN(abdctAng)*shankLength*COS(shankAng+thighAng)*zFTipDes;

DesireDriveForce_2 := TRUE;
END_METHOD

METHOD PUBLIC DownloadDriveCmds : BOOL
VAR_INPUT
	drive      : REFERENCE TO IntegratedDrive;
	driveIndex : INT;
	legIndex:UINT;
END_VAR
// the mapping between the angle of kinematics model and the angle of physical motor angle
(*motorAnglesOut[0]对应的是侧摆角，
motorAnglesOut[1]对应的是大腿角度
motorAnglesOut[2]对应的是小腿角度
但是驱动器0号对应小腿，所以将驱动器0赋值motorAnglesOut[2],即motorAnglesOut[phy2absMapping[driveIndex]],其中
phy2absMapping[0]=2
*)
IF legIndex=0 OR legIndex=5 THEN
	drive.SetImpdTarget(targetPos := motorAnglesOut[phy2absMapping[driveIndex]] - axisAngleOffset[phy2absMapping[driveIndex]], 
	                targetVel := motorAngVelOut[phy2absMapping[driveIndex]],
					additionalFce := jointTorqueOut[phy2absMapping[driveIndex]]);
ELSE
	drive.SetImpdTarget(targetPos := motorAnglesOut[phy2absMapping[driveIndex]], 
	                targetVel := motorAngVelOut[phy2absMapping[driveIndex]],
					additionalFce := jointTorqueOut[phy2absMapping[driveIndex]]);
END_IF
END_METHOD

METHOD PUBLIC ForwardKinetics : BOOL
VAR_INPUT
	motorAngles : ARRAY [0..2] OF LREAL;
	legIndex:INT;
END_VAR
VAR_OUTPUT
	tipPosition : ARRAY [0..2] OF LREAL;
END_VAR
VAR
	thighAng : LREAL;
	shankAng : LREAL;
	abductAng  : LREAL;
	xSagPlane : LREAL;
	ySagPlane : LREAL;
END_VAR
(*abductAng  := motorAngles[0];
thighAng := motorAngles[1];
shankAng := motorAngles[2];

xSagPlane := thighLength * COS(thighAng) + shankLength * COS(shankAng);
ySagPlane := thighLength * SIN(thighAng) + shankLength * SIN(shankAng);

tipPosition[0] := xSagPlane;
tipPosition[1] := COS(abductAng) * ySagPlane+SIN(abductAng) * sagPlaneOffset;
tipPosition[2] := SIN(abductAng) * ySagPlane-COS(abductAng) * sagPlaneOffset;*)
IF legIndex=0 OR legIndex=5 THEN
	gvl.legCtrl[legIndex].ForwardKinetics_1(motorAngles:=motorAngles  , tipPosition=> tipPosition);
ELSE
	gvl.legCtrl[legIndex].ForwardKinetics_2(motorAngles:=motorAngles  , tipPosition=> tipPosition);
END_IF

ForwardKinetics := TRUE;
END_METHOD

METHOD PUBLIC ForwardKinetics_1 : BOOL
VAR_INPUT
	motorAngles : ARRAY [0..2] OF LREAL;
END_VAR
VAR_OUTPUT
	tipPosition : ARRAY [0..2] OF LREAL;
END_VAR
VAR
	thighAng : LREAL;
	shankAng : LREAL;
	abductAng  : LREAL;
	xSagPlane : LREAL;
	ySagPlane : LREAL;
END_VAR
abductAng  := motorAngles[0];
thighAng := motorAngles[1];
shankAng := motorAngles[2];

xSagPlane := thighLength * COS(thighAng) + shankLength * COS(shankAng);
ySagPlane := thighLength * SIN(thighAng) + shankLength * SIN(shankAng);

tipPosition[0] := xSagPlane;
tipPosition[1] := COS(abductAng) * ySagPlane+SIN(abductAng) * sagPlaneOffset;
tipPosition[2] := SIN(abductAng) * ySagPlane-COS(abductAng) * sagPlaneOffset;

ForwardKinetics_1 := TRUE;
END_METHOD

METHOD PUBLIC ForwardKinetics_2 : BOOL
VAR_INPUT
	motorAngles : ARRAY [0..2] OF LREAL;
END_VAR
VAR_OUTPUT
	tipPosition : ARRAY [0..2] OF LREAL;
END_VAR
VAR
	thighAng : LREAL;
	shankAng : LREAL;
	abductAng  : LREAL;
	xSagPlane : LREAL;
	ySagPlane : LREAL;
END_VAR
abductAng  := motorAngles[0];
thighAng := motorAngles[1];
shankAng := motorAngles[2];

xSagPlane := thighLength * COS(thighAng) + shankLength * COS(shankAng+thighAng);
ySagPlane := thighLength * SIN(thighAng) + shankLength * SIN(shankAng+thighAng);

tipPosition[0] := xSagPlane;
tipPosition[1] := COS(abductAng) * ySagPlane+SIN(abductAng) * sagPlaneOffset;
tipPosition[2] := SIN(abductAng) * ySagPlane-COS(abductAng) * sagPlaneOffset;

ForwardKinetics_2 := TRUE;
END_METHOD

METHOD PUBLIC InitParam : BOOL
VAR_INPUT
	id            : UINT;
	shankLengthIn : LREAL;
	thighLengthIn : LREAL;
	sagPlaneOffsetIn:lreal;
END_VAR
legID       := id;
shankLength := shankLengthIn;
thighLength := thighLengthIn;
sagPlaneOffset:=sagPlaneOffsetIn;

InitParam := TRUE;
END_METHOD

METHOD PUBLIC InverseKinetics : BOOL
VAR_INPUT
	tipPosition : ARRAY [0..2] OF LREAL;
	refPosLast  : ARRAY[0..2] OF LREAL;
	legIndex:INT;
END_VAR
VAR_OUTPUT
	motorAngles : ARRAY [0..2] OF LREAL;
	isSingular  : BOOL;
END_VAR
VAR
	legSagAng : LREAL;
	legAbductAng : LREAL;
	legLength : LREAL;
	alpha     : LREAL;
	beta      : LREAL;
	x, y, z   : LREAL;
	xSag, ySag: LREAL;
	i: INT;
		
	motorAnglesAll:ARRAY[0..2,0..3] OF LREAL;
	theta:ARRAY[0..1] OF LREAL;
	phai:LREAL;
	t:LREAL;
	upper:ARRAY[0..2] OF LREAL:=[pi,2*pi,2*pi];
	lower:ARRAY[0..2] OF LREAL:=[-pi,0,0];
	j: INT;
END_VAR
(*x := tipPosition[0];
y := tipPosition[1];
z := tipPosition[2];
isSingular := FALSE;

phai:=atan2Fun(z,y);
t:=sagPlaneOffset/SQRT(y*y+z*z);
theta[0]:=phai+atan2Fun(t,SQRT(1-t*t));
theta[1]:=phai+atan2Fun(t,-SQRT(1-t*t));
FOR i:=0 TO 1 DO
	xSag:=x;
	ySag:=y*COS(theta[i])+z*SIN(theta[i]);
	legLength:=SQRT(xSag*xSag+ySag*ySag);
	legSagAng:=atan2Fun(ySag,xSag);
	alpha := ACOS((thighLength * thighLength + legLength * legLength - shankLength * shankLength) / 2.0 / thighLength / legLength);
	beta  := ACOS((thighLength * thighLength - legLength * legLength + shankLength * shankLength) / 2.0 / thighLength / shankLength);
	
	motorAnglesAll[0,0+2*i]:=theta[i];
	motorAnglesAll[1,0+2*i]:=legSagAng - alpha;
	motorAnglesAll[2,0+2*i]:= legSagAng - alpha + pi-beta;
	
	motorAnglesAll[0,1+2*i]:=theta[i];
	motorAnglesAll[1,1+2*i]:=legSagAng +alpha;
	motorAnglesAll[2,1+2*i]:= legSagAng + alpha - pi+beta;
END_FOR
FOR i:=0 TO 3 DO
	FOR j:=0 TO 2 DO
		motorAnglesAll[j,i]:=AngleCutFun(motorAnglesAll[j,i],upper[j],lower[j],2*pi);
	END_FOR
END_FOR

IF ABS(motorAnglesAll[0,0]-refPosLast[0])<ABS(motorAnglesAll[0,2]-refPosLast[0]) THEN
	IF ABS(motorAnglesAll[1,0]-refPosLast[1])<ABS(motorAnglesAll[1,1]-refPosLast[1]) THEN
		FOR j:=0 TO 2 DO
			motorAngles[j]:=motorAnglesAll[j,0];
		END_FOR
	ELSE
		FOR j:=0 TO 2 DO
			motorAngles[j]:=motorAnglesAll[j,1];
		END_FOR			
	END_IF
ELSE
	IF ABS(motorAnglesAll[1,2]-refPosLast[1])<ABS(motorAnglesAll[1,3]-refPosLast[1]) THEN
		FOR j:=0 TO 2 DO
			motorAngles[j]:=motorAnglesAll[j,2];
		END_FOR
	ELSE
		FOR j:=0 TO 2 DO
			motorAngles[j]:=motorAnglesAll[j,3];
		END_FOR			
	END_IF		
END_IF*)
IF legIndex=0 OR legIndex=5 THEN
	gvl.legCtrl[legIndex].InverseKinetics_1(tipPosition:=tipPosition , refPosLast:=refPosLast , motorAngles=>motorAngles , isSingular=>isSingular );
ELSE
	gvl.legCtrl[legIndex].InverseKinetics_2(tipPosition:=tipPosition , refPosLast:=refPosLast , motorAngles=>motorAngles , isSingular=>isSingular );
END_IF

InverseKinetics := isSingular;
END_METHOD

METHOD PUBLIC InverseKinetics_1 : BOOL
VAR_INPUT
	tipPosition : ARRAY [0..2] OF LREAL;
	refPosLast  : ARRAY[0..2] OF LREAL;
END_VAR
VAR_OUTPUT
	motorAngles : ARRAY [0..2] OF LREAL;
	isSingular  : BOOL;
END_VAR
VAR
	legSagAng : LREAL;
	legAbductAng : LREAL;
	legLength : LREAL;
	alpha     : LREAL;
	beta      : LREAL;
	x, y, z   : LREAL;
	xSag, ySag: LREAL;
	i: INT;
		
	motorAnglesAll:ARRAY[0..2,0..3] OF LREAL;
	theta:ARRAY[0..1] OF LREAL;
	phai:LREAL;
	t:LREAL;
	upper:ARRAY[0..2] OF LREAL:=[pi,2*pi,2*pi];
	lower:ARRAY[0..2] OF LREAL:=[-pi,0,0];
	j: INT;
END_VAR
x := tipPosition[0];
y := tipPosition[1];
z := tipPosition[2];
isSingular := FALSE;

phai:=atan2Fun(z,y);
t:=sagPlaneOffset/SQRT(y*y+z*z);
theta[0]:=phai+atan2Fun(t,SQRT(1-t*t));
theta[1]:=phai+atan2Fun(t,-SQRT(1-t*t));
FOR i:=0 TO 1 DO
	xSag:=x;
	ySag:=y*COS(theta[i])+z*SIN(theta[i]);
	legLength:=SQRT(xSag*xSag+ySag*ySag);
	legSagAng:=atan2Fun(ySag,xSag);
	alpha := ACOS((thighLength * thighLength + legLength * legLength - shankLength * shankLength) / 2.0 / thighLength / legLength);
	beta  := ACOS((thighLength * thighLength - legLength * legLength + shankLength * shankLength) / 2.0 / thighLength / shankLength);
	
	motorAnglesAll[0,0+2*i]:=theta[i];
	motorAnglesAll[1,0+2*i]:=legSagAng - alpha;
	motorAnglesAll[2,0+2*i]:= legSagAng - alpha + pi-beta;
	
	motorAnglesAll[0,1+2*i]:=theta[i];
	motorAnglesAll[1,1+2*i]:=legSagAng +alpha;
	motorAnglesAll[2,1+2*i]:= legSagAng + alpha - pi+beta;
END_FOR
FOR i:=0 TO 3 DO
	FOR j:=0 TO 2 DO
		motorAnglesAll[j,i]:=AngleCutFun(motorAnglesAll[j,i],upper[j],lower[j],2*pi);
	END_FOR
END_FOR

IF ABS(motorAnglesAll[0,0]-refPosLast[0])<ABS(motorAnglesAll[0,2]-refPosLast[0]) THEN
	IF ABS(motorAnglesAll[1,0]-refPosLast[1])<ABS(motorAnglesAll[1,1]-refPosLast[1]) THEN
		FOR j:=0 TO 2 DO
			motorAngles[j]:=motorAnglesAll[j,0];
		END_FOR
	ELSE
		FOR j:=0 TO 2 DO
			motorAngles[j]:=motorAnglesAll[j,1];
		END_FOR			
	END_IF
ELSE
	IF ABS(motorAnglesAll[1,2]-refPosLast[1])<ABS(motorAnglesAll[1,3]-refPosLast[1]) THEN
		FOR j:=0 TO 2 DO
			motorAngles[j]:=motorAnglesAll[j,2];
		END_FOR
	ELSE
		FOR j:=0 TO 2 DO
			motorAngles[j]:=motorAnglesAll[j,3];
		END_FOR			
	END_IF		
END_IF

InverseKinetics_1 := isSingular;
END_METHOD

METHOD PUBLIC InverseKinetics_2 : BOOL
VAR_INPUT
	tipPosition : ARRAY [0..2] OF LREAL;
	refPosLast  : ARRAY[0..2] OF LREAL;
END_VAR
VAR_OUTPUT
	motorAngles : ARRAY [0..2] OF LREAL;
	isSingular  : BOOL;
END_VAR
VAR
	legSagAng : LREAL;
	legAbductAng : LREAL;
	legLength : LREAL;
	alpha     : LREAL;
	beta      : LREAL;
	x, y, z   : LREAL;
	xSag, ySag: LREAL;
	i: INT;
		
	motorAnglesAll:ARRAY[0..2,0..3] OF LREAL;
	theta:ARRAY[0..1] OF LREAL;
	phai:LREAL;
	t:LREAL;
	upper:ARRAY[0..2] OF LREAL:=[pi,2*pi,2*pi];
	lower:ARRAY[0..2] OF LREAL:=[-pi,0,0];
	j: INT;
	refPosLastModel:ARRAY[0..2] OF LREAL;
END_VAR
x := tipPosition[0];
y := tipPosition[1];
z := tipPosition[2];
isSingular := FALSE;

phai:=atan2Fun(z,y);
t:=sagPlaneOffset/SQRT(y*y+z*z);
theta[0]:=phai+atan2Fun(t,SQRT(1-t*t));
theta[1]:=phai+atan2Fun(t,-SQRT(1-t*t));
FOR i:=0 TO 1 DO
	xSag:=x;
	ySag:=y*COS(theta[i])+z*SIN(theta[i]);
	legLength:=SQRT(xSag*xSag+ySag*ySag);
	legSagAng:=atan2Fun(ySag,xSag);
	alpha := ACOS((thighLength * thighLength + legLength * legLength - shankLength * shankLength) / 2.0 / thighLength / legLength);
	beta  := ACOS((thighLength * thighLength - legLength * legLength + shankLength * shankLength) / 2.0 / thighLength / shankLength);
	
	motorAnglesAll[0,0+2*i]:=theta[i];
	motorAnglesAll[1,0+2*i]:=legSagAng - alpha;
	motorAnglesAll[2,0+2*i]:= legSagAng - alpha + pi-beta;
	
	motorAnglesAll[0,1+2*i]:=theta[i];
	motorAnglesAll[1,1+2*i]:=legSagAng +alpha;
	motorAnglesAll[2,1+2*i]:= legSagAng + alpha - pi+beta;
END_FOR
FOR i:=0 TO 3 DO
	FOR j:=0 TO 2 DO
		motorAnglesAll[j,i]:=AngleCutFun(motorAnglesAll[j,i],upper[j],lower[j],2*pi);
	END_FOR
END_FOR

refPosLastModel[0]:=refPosLast[0];
refPosLastModel[1]:=AngleCutFun(refPosLast[1],2*pi,0,2*pi);
refPosLastModel[2]:=AngleCutFun(refPosLast[1]+refPosLast[2],2*pi,0,2*pi);


IF ABS(motorAnglesAll[0,0]-refPosLastModel[0])<ABS(motorAnglesAll[0,2]-refPosLastModel[0]) THEN
	IF Min3Value(ABS(motorAnglesAll[1,0]-refPosLastModel[1]),ABS(motorAnglesAll[1,0]+2*pi-refPosLastModel[1]),ABS(motorAnglesAll[1,0]-2*pi-refPosLastModel[1]))
       <Min3Value(ABS(motorAnglesAll[1,1]-refPosLastModel[1]),ABS(motorAnglesAll[1,1]+2*pi-refPosLastModel[1]),ABS(motorAnglesAll[1,1]-2*pi-refPosLastModel[1])) THEN
		FOR j:=0 TO 2 DO
			motorAngles[j]:=motorAnglesAll[j,0];
		END_FOR
	ELSE
		FOR j:=0 TO 2 DO
			motorAngles[j]:=motorAnglesAll[j,1];
		END_FOR			
	END_IF
ELSE
	IF Min3Value(ABS(motorAnglesAll[1,2]-refPosLastModel[1]),ABS(motorAnglesAll[1,2]+2*pi-refPosLastModel[1]),ABS(motorAnglesAll[1,2]-2*pi-refPosLastModel[1]))
       <Min3Value(ABS(motorAnglesAll[1,3]-refPosLastModel[1]),ABS(motorAnglesAll[1,3]+2*pi-refPosLastModel[1]),ABS(motorAnglesAll[1,3]-2*pi-refPosLastModel[1])) THEN
		FOR j:=0 TO 2 DO
			motorAngles[j]:=motorAnglesAll[j,2];
		END_FOR
	ELSE
		FOR j:=0 TO 2 DO
			motorAngles[j]:=motorAnglesAll[j,3];
		END_FOR			
	END_IF		
END_IF

motorAngles[1]:=MinDistanceValue(motorAngles[1],refPosLastModel[1]);
motorAngles[2]:=MinDistanceValue(motorAngles[2],refPosLastModel[2]);

motorAngles[2]:=MinDistanceValue(motorAngles[2]-motorAngles[1],refPosLast[2]);
motorAngles[1]:=MinDistanceValue(motorAngles[1],refPosLast[1]);



(*motorAngles[2]:=Min3Value(ABS(motorAngles[2]-refPosLastModel[2]),ABS(motorAngles[2]+2*pi-refPosLastModel[2]),ABS(motorAngles[2]-2*pi-refPosLastModel[2]))+refPosLastModel[2];

motorAngles[2]:=Min3Value(motorAngles[2]-motorAngles[1]-refPosLast[2],motorAngles[2]-motorAngles[1]+2*pi-refPosLast[2],motorAngles[2]-motorAngles[1]-2*pi-refPosLast[2])+refPosLast[2];

motorAngles[1]:=Min3Value(motorAngles[1]-refPosLast[1],motorAngles[1]+2*pi-refPosLast[1],motorAngles[1]-2*pi-refPosLast[1])+refPosLast[1];*)

//motorAngles[2]:=motorAngles[2]-motorAngles[1];

InverseKinetics_2 := isSingular;
END_METHOD

METHOD PUBLIC InversePosAndVel : BOOL
VAR_INPUT
	tipPos : ARRAY[0..2] OF LREAL;
	tipVel : ARRAY[0..2] OF LREAL;
	refPosLast  : ARRAY[0..2] OF LREAL;
	legIndex:INT;
END_VAR
VAR_OUTPUT
	jntPos : ARRAY[0..2] OF LREAL;
	jntVel : ARRAY[0..2] OF LREAL; 
END_VAR
VAR	
	legSagAng : LREAL;
	legAbductAng : LREAL;
	legLength : LREAL;
	alpha     : LREAL;
	beta      : LREAL;
	x, y, z   : LREAL;
	xSag, ySag: LREAL;
	i: INT;
		
	motorAnglesAll:ARRAY[0..2,0..3] OF LREAL;
	theta:ARRAY[0..1] OF LREAL;
	phai:LREAL;
	t:LREAL;
	upper:ARRAY[0..2] OF LREAL:=[pi,2*pi,2*pi];
	lower:ARRAY[0..2] OF LREAL:=[-pi,0,0];
	j: INT;
	theta_a,theta_t,theta_s,csc:LREAL;
END_VAR
(*x := tipPos[0];
y := tipPos[1];
z := tipPos[2];

phai:=atan2Fun(z,y);
t:=sagPlaneOffset/SQRT(y*y+z*z);
theta[0]:=phai+atan2Fun(t,SQRT(1-t*t));
theta[1]:=phai+atan2Fun(t,-SQRT(1-t*t));
FOR i:=0 TO 1 DO
	xSag:=x;
	ySag:=y*COS(theta[i])+z*SIN(theta[i]);
	legLength:=SQRT(xSag*xSag+ySag*ySag);
	legSagAng:=atan2Fun(ySag,xSag);
	alpha := ACOS((thighLength * thighLength + legLength * legLength - shankLength * shankLength) / 2.0 / thighLength / legLength);
	beta  := ACOS((thighLength * thighLength - legLength * legLength + shankLength * shankLength) / 2.0 / thighLength / shankLength);
	
	motorAnglesAll[0,0+2*i]:=theta[i];
	motorAnglesAll[1,0+2*i]:=legSagAng - alpha;
	motorAnglesAll[2,0+2*i]:= legSagAng - alpha + pi-beta;
	
	motorAnglesAll[0,1+2*i]:=theta[i];
	motorAnglesAll[1,1+2*i]:=legSagAng +alpha;
	motorAnglesAll[2,1+2*i]:= legSagAng + alpha - pi+beta;
END_FOR
FOR i:=0 TO 3 DO
	FOR j:=0 TO 2 DO
		motorAnglesAll[j,i]:=AngleCutFun(motorAnglesAll[j,i],upper[j],lower[j],2*pi);
	END_FOR
END_FOR

IF ABS(motorAnglesAll[0,0]-refPosLast[0])<ABS(motorAnglesAll[0,2]-refPosLast[0]) THEN
	IF ABS(motorAnglesAll[1,0]-refPosLast[1])<ABS(motorAnglesAll[1,1]-refPosLast[1]) THEN
		FOR j:=0 TO 2 DO
			jntPos[j]:=motorAnglesAll[j,0];
		END_FOR
	ELSE
		FOR j:=0 TO 2 DO
			jntPos[j]:=motorAnglesAll[j,1];
		END_FOR			
	END_IF
ELSE
	IF ABS(motorAnglesAll[1,2]-refPosLast[1])<ABS(motorAnglesAll[1,3]-refPosLast[1]) THEN
		FOR j:=0 TO 2 DO
			jntPos[j]:=motorAnglesAll[j,2];
		END_FOR
	ELSE
		FOR j:=0 TO 2 DO
			jntPos[j]:=motorAnglesAll[j,3];
		END_FOR			
	END_IF		
END_IF
theta_a:=jntPos[0];
theta_t:=jntPos[1];
theta_s:=jntPos[2];
csc:=1/SIN(theta_s-theta_t);
ySag:=thighLength*SIN(theta_t)+shankLength*SIN(theta_s);

jntVel[0]:=-SIN(theta_a)/ySag*tipVel[1]+COS(theta_a)/ySag*tipVel[2];
jntVel[1]:=COS(theta_s)*csc/thighLength*tipVel[0]+SIN(theta_s)*(sagPlaneOffset*SIN(theta_a)+ySag*COS(theta_a))*csc/(thighLength*ySag)*tipVel[1]-SIN(theta_s)*(sagPlaneOffset*COS(theta_a)-ySag*SIN(theta_a))*csc/(thighLength*ySag)*tipVel[2];
jntVel[2]:=-COS(theta_t)*csc/shankLength*tipVel[0]-SIN(theta_t)*(sagPlaneOffset*SIN(theta_a)+ySag*COS(theta_a))*csc/(shankLength*ySag)*tipVel[1]+SIN(theta_t)*(sagPlaneOffset*COS(theta_a)-ySag*SIN(theta_a))*csc/(shankLength*ySag)*tipVel[2];     
*)
IF legIndex=0 OR legIndex=5 THEN
	gvl.legCtrl[legIndex].InversePosAndVel_1(tipPos:=tipPos  , tipVel:= tipVel, refPosLast:=refPosLast , jntPos=> jntPos, jntVel=>jntVel );
ELSE
	gvl.legCtrl[legIndex].InversePosAndVel_2(tipPos:=tipPos  , tipVel:= tipVel, refPosLast:=refPosLast , jntPos=> jntPos, jntVel=>jntVel );
END_IF
END_METHOD

METHOD PUBLIC InversePosAndVel_1 : BOOL
VAR_INPUT
	tipPos : ARRAY[0..2] OF LREAL;
	tipVel : ARRAY[0..2] OF LREAL;
	refPosLast  : ARRAY[0..2] OF LREAL;
END_VAR
VAR_OUTPUT
	jntPos : ARRAY[0..2] OF LREAL;
	jntVel : ARRAY[0..2] OF LREAL; 
END_VAR
VAR	
	legSagAng : LREAL;
	legAbductAng : LREAL;
	legLength : LREAL;
	alpha     : LREAL;
	beta      : LREAL;
	x, y, z   : LREAL;
	xSag, ySag: LREAL;
	i: INT;
		
	motorAnglesAll:ARRAY[0..2,0..3] OF LREAL;
	theta:ARRAY[0..1] OF LREAL;
	phai:LREAL;
	t:LREAL;
	upper:ARRAY[0..2] OF LREAL:=[pi,2*pi,2*pi];
	lower:ARRAY[0..2] OF LREAL:=[-pi,0,0];
	j: INT;
	theta_a,theta_t,theta_s,csc:LREAL;
END_VAR
x := tipPos[0];
y := tipPos[1];
z := tipPos[2];

phai:=atan2Fun(z,y);
t:=sagPlaneOffset/SQRT(y*y+z*z);
theta[0]:=phai+atan2Fun(t,SQRT(1-t*t));
theta[1]:=phai+atan2Fun(t,-SQRT(1-t*t));
FOR i:=0 TO 1 DO
	xSag:=x;
	ySag:=y*COS(theta[i])+z*SIN(theta[i]);
	legLength:=SQRT(xSag*xSag+ySag*ySag);
	legSagAng:=atan2Fun(ySag,xSag);
	alpha := ACOS((thighLength * thighLength + legLength * legLength - shankLength * shankLength) / 2.0 / thighLength / legLength);
	beta  := ACOS((thighLength * thighLength - legLength * legLength + shankLength * shankLength) / 2.0 / thighLength / shankLength);
	
	motorAnglesAll[0,0+2*i]:=theta[i];
	motorAnglesAll[1,0+2*i]:=legSagAng - alpha;
	motorAnglesAll[2,0+2*i]:= legSagAng - alpha + pi-beta;
	
	motorAnglesAll[0,1+2*i]:=theta[i];
	motorAnglesAll[1,1+2*i]:=legSagAng +alpha;
	motorAnglesAll[2,1+2*i]:= legSagAng + alpha - pi+beta;
END_FOR
FOR i:=0 TO 3 DO
	FOR j:=0 TO 2 DO
		motorAnglesAll[j,i]:=AngleCutFun(motorAnglesAll[j,i],upper[j],lower[j],2*pi);
	END_FOR
END_FOR

IF ABS(motorAnglesAll[0,0]-refPosLast[0])<ABS(motorAnglesAll[0,2]-refPosLast[0]) THEN
	IF ABS(motorAnglesAll[1,0]-refPosLast[1])<ABS(motorAnglesAll[1,1]-refPosLast[1]) THEN
		FOR j:=0 TO 2 DO
			jntPos[j]:=motorAnglesAll[j,0];
		END_FOR
	ELSE
		FOR j:=0 TO 2 DO
			jntPos[j]:=motorAnglesAll[j,1];
		END_FOR			
	END_IF
ELSE
	IF ABS(motorAnglesAll[1,2]-refPosLast[1])<ABS(motorAnglesAll[1,3]-refPosLast[1]) THEN
		FOR j:=0 TO 2 DO
			jntPos[j]:=motorAnglesAll[j,2];
		END_FOR
	ELSE
		FOR j:=0 TO 2 DO
			jntPos[j]:=motorAnglesAll[j,3];
		END_FOR			
	END_IF		
END_IF
theta_a:=jntPos[0];
theta_t:=jntPos[1];
theta_s:=jntPos[2];
csc:=1/SIN(theta_s-theta_t);
ySag:=thighLength*SIN(theta_t)+shankLength*SIN(theta_s);

jntVel[0]:=-SIN(theta_a)/ySag*tipVel[1]+COS(theta_a)/ySag*tipVel[2];
jntVel[1]:=COS(theta_s)*csc/thighLength*tipVel[0]+SIN(theta_s)*(sagPlaneOffset*SIN(theta_a)+ySag*COS(theta_a))*csc/(thighLength*ySag)*tipVel[1]-SIN(theta_s)*(sagPlaneOffset*COS(theta_a)-ySag*SIN(theta_a))*csc/(thighLength*ySag)*tipVel[2];
jntVel[2]:=-COS(theta_t)*csc/shankLength*tipVel[0]-SIN(theta_t)*(sagPlaneOffset*SIN(theta_a)+ySag*COS(theta_a))*csc/(shankLength*ySag)*tipVel[1]+SIN(theta_t)*(sagPlaneOffset*COS(theta_a)-ySag*SIN(theta_a))*csc/(shankLength*ySag)*tipVel[2];
END_METHOD

METHOD PUBLIC InversePosAndVel_2 : BOOL
VAR_INPUT
	tipPos : ARRAY[0..2] OF LREAL;
	tipVel : ARRAY[0..2] OF LREAL;
	refPosLast  : ARRAY[0..2] OF LREAL;
END_VAR
VAR_OUTPUT
	jntPos : ARRAY[0..2] OF LREAL;
	jntVel : ARRAY[0..2] OF LREAL; 
END_VAR
VAR	
	legSagAng : LREAL;
	legAbductAng : LREAL;
	legLength : LREAL;
	alpha     : LREAL;
	beta      : LREAL;
	x, y, z   : LREAL;
	xSag, ySag: LREAL;
	i: INT;
		
	motorAnglesAll:ARRAY[0..2,0..3] OF LREAL;
	theta:ARRAY[0..1] OF LREAL;
	phai:LREAL;
	t:LREAL;
	upper:ARRAY[0..2] OF LREAL:=[pi,2*pi,2*pi];
	lower:ARRAY[0..2] OF LREAL:=[-pi,0,0];
	j: INT;
	theta_a,theta_t,theta_s,csc:LREAL;
	refPosLastModel:ARRAY[0..2] OF LREAL;
	motorAngles : ARRAY [0..2] OF LREAL;
END_VAR
x := tipPos[0];
y := tipPos[1];
z := tipPos[2];

phai:=atan2Fun(z,y);
t:=sagPlaneOffset/SQRT(y*y+z*z);
theta[0]:=phai+atan2Fun(t,SQRT(1-t*t));
theta[1]:=phai+atan2Fun(t,-SQRT(1-t*t));
FOR i:=0 TO 1 DO
	xSag:=x;
	ySag:=y*COS(theta[i])+z*SIN(theta[i]);
	legLength:=SQRT(xSag*xSag+ySag*ySag);
	legSagAng:=atan2Fun(ySag,xSag);
	alpha := ACOS((thighLength * thighLength + legLength * legLength - shankLength * shankLength) / 2.0 / thighLength / legLength);
	beta  := ACOS((thighLength * thighLength - legLength * legLength + shankLength * shankLength) / 2.0 / thighLength / shankLength);
	
	motorAnglesAll[0,0+2*i]:=theta[i];
	motorAnglesAll[1,0+2*i]:=legSagAng - alpha;
	motorAnglesAll[2,0+2*i]:= legSagAng - alpha + pi-beta;
	
	motorAnglesAll[0,1+2*i]:=theta[i];
	motorAnglesAll[1,1+2*i]:=legSagAng +alpha;
	motorAnglesAll[2,1+2*i]:= legSagAng + alpha - pi+beta;
END_FOR
FOR i:=0 TO 3 DO
	FOR j:=0 TO 2 DO
		motorAnglesAll[j,i]:=AngleCutFun(motorAnglesAll[j,i],upper[j],lower[j],2*pi);
	END_FOR
END_FOR

refPosLastModel[0]:=refPosLast[0];
refPosLastModel[1]:=AngleCutFun(refPosLast[1],2*pi,0,2*pi);
refPosLastModel[2]:=AngleCutFun(refPosLast[1]+refPosLast[2],2*pi,0,2*pi);

IF ABS(motorAnglesAll[0,0]-refPosLastModel[0])<ABS(motorAnglesAll[0,2]-refPosLastModel[0]) THEN
	IF Min3Value(ABS(motorAnglesAll[1,0]-refPosLastModel[1]),ABS(motorAnglesAll[1,0]+2*pi-refPosLastModel[1]),ABS(motorAnglesAll[1,0]-2*pi-refPosLastModel[1]))
       <Min3Value(ABS(motorAnglesAll[1,1]-refPosLastModel[1]),ABS(motorAnglesAll[1,1]+2*pi-refPosLastModel[1]),ABS(motorAnglesAll[1,1]-2*pi-refPosLastModel[1])) THEN
		FOR j:=0 TO 2 DO
			motorAngles[j]:=motorAnglesAll[j,0];
		END_FOR
	ELSE
		FOR j:=0 TO 2 DO
			motorAngles[j]:=motorAnglesAll[j,1];
		END_FOR			
	END_IF
ELSE
	IF Min3Value(ABS(motorAnglesAll[1,2]-refPosLastModel[1]),ABS(motorAnglesAll[1,2]+2*pi-refPosLastModel[1]),ABS(motorAnglesAll[1,2]-2*pi-refPosLastModel[1]))
       <Min3Value(ABS(motorAnglesAll[1,3]-refPosLastModel[1]),ABS(motorAnglesAll[1,3]+2*pi-refPosLastModel[1]),ABS(motorAnglesAll[1,3]-2*pi-refPosLastModel[1])) THEN
		FOR j:=0 TO 2 DO
			motorAngles[j]:=motorAnglesAll[j,2];
		END_FOR
	ELSE
		FOR j:=0 TO 2 DO
			motorAngles[j]:=motorAnglesAll[j,3];
		END_FOR			
	END_IF		
END_IF



theta_a:=motorAngles[0];
theta_t:=motorAngles[1];
theta_s:=motorAngles[2];
csc:=1/SIN(theta_s-theta_t);
ySag:=thighLength*SIN(theta_t)+shankLength*SIN(theta_s);

jntVel[0]:=-SIN(theta_a)/ySag*tipVel[1]+COS(theta_a)/ySag*tipVel[2];
jntVel[1]:=COS(theta_s)*csc/thighLength*tipVel[0]+SIN(theta_s)*(sagPlaneOffset*SIN(theta_a)+ySag*COS(theta_a))*csc/(thighLength*ySag)*tipVel[1]-SIN(theta_s)*(sagPlaneOffset*COS(theta_a)-ySag*SIN(theta_a))*csc/(thighLength*ySag)*tipVel[2];
jntVel[2]:=-COS(theta_t)*csc/shankLength*tipVel[0]-SIN(theta_t)*(sagPlaneOffset*SIN(theta_a)+ySag*COS(theta_a))*csc/(shankLength*ySag)*tipVel[1]+SIN(theta_t)*(sagPlaneOffset*COS(theta_a)-ySag*SIN(theta_a))*csc/(shankLength*ySag)*tipVel[2];     

motorAngles[1]:=MinDistanceValue(motorAngles[1],refPosLastModel[1]);
motorAngles[2]:=MinDistanceValue(motorAngles[2],refPosLastModel[2]);

motorAngles[2]:=MinDistanceValue(motorAngles[2]-motorAngles[1],refPosLast[2]);
motorAngles[1]:=MinDistanceValue(motorAngles[1],refPosLast[1]);

jntPos[0]:=motorAngles[0];
jntPos[1]:=motorAngles[1];
jntPos[2]:=motorAngles[2];

jntVel[2]:=jntVel[2]- jntVel[1];
END_METHOD

METHOD PUBLIC SetReference : BOOL
VAR_INPUT
END_VAR
VAR
	j: INT;
END_VAR
FOR j := 0 TO 2 DO
	motorAnglesOut[j] := gvl.jntRefPos[legId, j];
	motorAngVelOut[j] := gvl.jntRefVel[legId, j];
	jointTorqueOut[j] := gvl.jntRefFce[legId, j];
END_FOR
END_METHOD

METHOD PUBLIC TipForce : BOOL
VAR_INPUT
	motorTrq : ARRAY[0..2] OF LREAL;
	motorAng : ARRAY[0..2] OF LREAL;
	legIndex:INT;
END_VAR
VAR_OUTPUT
	tipFce : ARRAY[0..2] OF LREAL;
END_VAR
VAR
	thighTrq : LREAL;
	shankTrq : LREAL;
	abdctTrq : LREAL;
	thighAng : LREAL;
	shankAng : LREAL;
	abdctAng : LREAL;
	
	ySag     : LREAL;
	csc      : LREAL;
END_VAR
(*abdctTrq := motorTrq[0];
thighTrq := motorTrq[1];
shankTrq := motorTrq[2];

abdctAng := motorAng[0];
thighAng := motorAng[1];
shankAng := motorAng[2];

ySag := thighLength*SIN(thighAng) + shankLength*SIN(shankAng);
csc := (1/SIN(shankAng-thighAng));

tipFce[0] :=  csc / thighLength * COS(shankAng) * thighTrq - csc / shankLength * COS(thighAng) * shankTrq;
tipFce[1]:=  -SIN(abdctAng)/ySag * abdctTrq + SIN(shankAng)*(sagPlaneOffset*SIN(abdctAng)+ySag*COS(abdctAng))*csc/(thighLength*ySag)*thighTrq - SIN(thighAng)*(sagPlaneOffset*SIN(abdctAng)+ySag*COS(abdctAng))*csc/(shankLength*ySag)* shankTrq;
tipFce[2]:=   COS(abdctAng)/ySag * abdctTrq - SIN(shankAng)*(sagPlaneOffset*COS(abdctAng)-ySag*SIN(abdctAng))*csc/(thighLength*ySag) * thighTrq + SIN(thighAng)*(sagPlaneOffset*COS(abdctAng)-ySag*SIN(abdctAng))*csc/(shankLength*ySag) * shankTrq;
*)
IF legIndex=0 OR legIndex=5 THEN
	gvl.legCtrl[legIndex].TipForce_1(motorTrq:=motorTrq  , motorAng:=motorAng  , tipFce=>tipFce );
ELSE
	gvl.legCtrl[legIndex].TipForce_2(motorTrq:=motorTrq  , motorAng:=motorAng  , tipFce=>tipFce );
END_IF

TipForce := TRUE;
END_METHOD

METHOD PUBLIC TipForce_1 : BOOL
VAR_INPUT
	motorTrq : ARRAY[0..2] OF LREAL;
	motorAng : ARRAY[0..2] OF LREAL;
END_VAR
VAR_OUTPUT
	tipFce : ARRAY[0..2] OF LREAL;
END_VAR
VAR
	thighTrq : LREAL;
	shankTrq : LREAL;
	abdctTrq : LREAL;
	thighAng : LREAL;
	shankAng : LREAL;
	abdctAng : LREAL;
	
	ySag     : LREAL;
	csc      : LREAL;
END_VAR
abdctTrq := motorTrq[0];
thighTrq := motorTrq[1];
shankTrq := motorTrq[2];

abdctAng := motorAng[0];
thighAng := motorAng[1];
shankAng := motorAng[2];

ySag := thighLength*SIN(thighAng) + shankLength*SIN(shankAng);
csc := (1/SIN(shankAng-thighAng));

tipFce[0] :=  csc / thighLength * COS(shankAng) * thighTrq - csc / shankLength * COS(thighAng) * shankTrq;
tipFce[1]:=  -SIN(abdctAng)/ySag * abdctTrq + SIN(shankAng)*(sagPlaneOffset*SIN(abdctAng)+ySag*COS(abdctAng))*csc/(thighLength*ySag)*thighTrq - SIN(thighAng)*(sagPlaneOffset*SIN(abdctAng)+ySag*COS(abdctAng))*csc/(shankLength*ySag)* shankTrq;
tipFce[2]:=   COS(abdctAng)/ySag * abdctTrq - SIN(shankAng)*(sagPlaneOffset*COS(abdctAng)-ySag*SIN(abdctAng))*csc/(thighLength*ySag) * thighTrq + SIN(thighAng)*(sagPlaneOffset*COS(abdctAng)-ySag*SIN(abdctAng))*csc/(shankLength*ySag) * shankTrq;

TipForce_1 := TRUE;
END_METHOD

METHOD PUBLIC TipForce_2 : BOOL
VAR_INPUT
	motorTrq : ARRAY[0..2] OF LREAL;
	motorAng : ARRAY[0..2] OF LREAL;
END_VAR
VAR_OUTPUT
	tipFce : ARRAY[0..2] OF LREAL;
END_VAR
VAR
	thighTrq : LREAL;
	shankTrq : LREAL;
	abdctTrq : LREAL;
	thighAng : LREAL;
	shankAng : LREAL;
	abdctAng : LREAL;
	
	ySag     : LREAL;
	csc      : LREAL;
END_VAR
abdctTrq := motorTrq[0];
thighTrq := motorTrq[1];
shankTrq := motorTrq[2];

abdctAng := motorAng[0];
thighAng := motorAng[1];
shankAng := motorAng[2];

ySag := thighLength*SIN(thighAng) + shankLength*SIN(shankAng+thighAng);
csc := 1/SIN(shankAng);

tipFce[0] :=  csc / thighLength * COS(shankAng+thighAng) * thighTrq - csc / shankLength * COS(thighAng) * shankTrq- csc / thighLength * COS(thighAng+shankAng) * shankTrq;
tipFce[1]:=  -SIN(abdctAng)/ySag * abdctTrq + SIN(shankAng+thighAng)*(sagPlaneOffset*SIN(abdctAng)+ySag*COS(abdctAng))*csc/(thighLength*ySag)*thighTrq - (sagPlaneOffset*SIN(abdctAng)+ySag*COS(abdctAng))*csc*(SIN(thighAng)/(shankLength*ySag)+SIN(thighAng+shankAng)/(thighLength*ySag))* shankTrq;
tipFce[2]:=   COS(abdctAng)/ySag * abdctTrq - SIN(shankAng+thighAng)*(sagPlaneOffset*COS(abdctAng)-ySag*SIN(abdctAng))*csc/(thighLength*ySag) * thighTrq + (sagPlaneOffset*COS(abdctAng)-ySag*SIN(abdctAng))*csc*(SIN(thighAng)/(shankLength*ySag)+SIN(thighAng+shankAng)/(thighLength*ySag)) * shankTrq;

TipForce_2 := TRUE;
END_METHOD

METHOD PUBLIC TipVelocity : BOOL
VAR_INPUT
	motorVel : ARRAY[0..2] OF LREAL;
	motorAng : ARRAY[0..2] OF LREAL;
	legIndex:INT;
END_VAR
VAR_OUTPUT
	tipVel : ARRAY[0..2] OF LREAL;
END_VAR
VAR
	thighVel : LREAL;
	shankVel : LREAL;
	abductVel: LREAL;
	thighAng : LREAL;
	shankAng : LREAL;
	abductAng: LREAL;
	
	ySag     : LREAL;
	ySagVel  : LREAL;
END_VAR
(*abductVel := motorVel[0];
thighVel  := motorVel[1];
shankVel  := motorVel[2];

abductAng := motorAng[0];
thighAng  := motorAng[1];
shankAng  := motorAng[2];

ySag      := thighLength*SIN(thighAng) + shankLength*SIN(shankAng);
ySagVel   := thighLength * COS(thighAng) * thighVel + shankLength * COS(shankAng) * shankVel;

tipVel[0] := -thighLength * SIN(thighAng) * thighVel - shankLength * SIN(shankAng) * shankVel;
tipVel[1] :=  COS(abductAng)*ySagVel - SIN(abductAng) * ySag * abductVel+COS(abductAng)*sagPlaneOffset*abductVel;
tipVel[2] :=  SIN(abductAng)*ySagVel + COS(abductAng) * ySag * abductVel+SIN(abductAng)*sagPlaneOffset*abductVel;*)
IF legIndex=0 OR legIndex=5 THEN
	gvl.legCtrl[legIndex].TipVelocity_1(motorVel:= motorVel, motorAng:=motorAng  , tipVel=> tipVel);
ELSE
	gvl.legCtrl[legIndex].TipVelocity_2(motorVel:= motorVel, motorAng:=motorAng  , tipVel=> tipVel);
END_IF

TipVelocity := TRUE;
END_METHOD

METHOD PUBLIC TipVelocity_1 : BOOL
VAR_INPUT
	motorVel : ARRAY[0..2] OF LREAL;
	motorAng : ARRAY[0..2] OF LREAL;
END_VAR
VAR_OUTPUT
	tipVel : ARRAY[0..2] OF LREAL;
END_VAR
VAR
	thighVel : LREAL;
	shankVel : LREAL;
	abductVel: LREAL;
	thighAng : LREAL;
	shankAng : LREAL;
	abductAng: LREAL;
	
	ySag     : LREAL;
	ySagVel  : LREAL;
END_VAR
abductVel := motorVel[0];
thighVel  := motorVel[1];
shankVel  := motorVel[2];

abductAng := motorAng[0];
thighAng  := motorAng[1];
shankAng  := motorAng[2];

ySag      := thighLength*SIN(thighAng) + shankLength*SIN(shankAng);
ySagVel   := thighLength * COS(thighAng) * thighVel + shankLength * COS(shankAng) * shankVel;

tipVel[0] := -thighLength * SIN(thighAng) * thighVel - shankLength * SIN(shankAng) * shankVel;
tipVel[1] :=  COS(abductAng)*ySagVel - SIN(abductAng) * ySag * abductVel+COS(abductAng)*sagPlaneOffset*abductVel;
tipVel[2] :=  SIN(abductAng)*ySagVel + COS(abductAng) * ySag * abductVel+sin(abductAng)*sagPlaneOffset*abductVel;

TipVelocity_1 := TRUE;
END_METHOD

METHOD PUBLIC TipVelocity_2 : BOOL
VAR_INPUT
	motorVel : ARRAY[0..2] OF LREAL;
	motorAng : ARRAY[0..2] OF LREAL;
END_VAR
VAR_OUTPUT
	tipVel : ARRAY[0..2] OF LREAL;
END_VAR
VAR
	thighVel : LREAL;
	shankVel : LREAL;
	abductVel: LREAL;
	thighAng : LREAL;
	shankAng : LREAL;
	abductAng: LREAL;
	
	ySag     : LREAL;
	ySagVel  : LREAL;
END_VAR
abductVel := motorVel[0];
thighVel  := motorVel[1];
shankVel  := motorVel[2];

abductAng := motorAng[0];
thighAng  := motorAng[1];
shankAng  := motorAng[2];

ySag      := thighLength*SIN(thighAng) + shankLength*SIN(shankAng+thighAng);
ySagVel   := (thighLength * COS(thighAng)+shankLength*COS(shankAng+thighAng)) * thighVel + shankLength * COS(shankAng+thighAng) * shankVel;

tipVel[0] := -(thighLength * SIN(thighAng)+shankLength*SIN(shankAng+thighAng)) * thighVel - shankLength * SIN(shankAng+thighAng) * shankVel;
tipVel[1] :=  COS(abductAng)*ySagVel - SIN(abductAng) * ySag * abductVel+COS(abductAng)*sagPlaneOffset*abductVel;
tipVel[2] :=  SIN(abductAng)*ySagVel + COS(abductAng) * ySag * abductVel+sin(abductAng)*sagPlaneOffset*abductVel;

TipVelocity_2 := TRUE;
END_METHOD

METHOD PUBLIC UpdateDriveFeedbacks : BOOL
VAR_INPUT
	drive      : REFERENCE TO IntegratedDrive;
	//drive_second      : REFERENCE TO IntegratedDrive;
	driveIndex : UINT;//0->shank,1->thigh,2->side
	legIndex:INT;
END_VAR
// the mapping between the angle of kinematics model and the angle of physical motor angle
//0号驱动器对应小腿，1号对应大腿，2号对应侧摆
(*motorAnglesIn[phy2absMapping[driveIndex]] := drive.motorAngle + axisAngleOffset[phy2absMapping[driveIndex]];//当前实际位置，运动学输入
motorAngVelIn[phy2absMapping[driveIndex]] := drive.motorAngVel;
jointTorqueIn[phy2absMapping[driveIndex]] := drive.trqCalibrated;
motorRefAnglesIn[phy2absMapping[driveIndex]] := drive.tgtAngle + axisAngleOffset[phy2absMapping[driveIndex]];//当前参考角度，运动学输入*)

IF legIndex=0 OR legIndex=5 THEN
	motorAnglesIn[phy2absMapping[driveIndex]] := drive.motorAngle + axisAngleOffset[phy2absMapping[driveIndex]];//当前实际位置，运动学输入
	motorAngVelIn[phy2absMapping[driveIndex]] := drive.motorAngVel;
	jointTorqueIn[phy2absMapping[driveIndex]] := drive.trqCalibrated;
	motorRefAnglesIn[phy2absMapping[driveIndex]] := drive.tgtAngle + axisAngleOffset[phy2absMapping[driveIndex]];//当前参考角度，运动学输入
ELSE
	motorAnglesIn[phy2absMapping[driveIndex]] := drive.motorAngle ;//当前实际位置，运动学输入
	motorAngVelIn[phy2absMapping[driveIndex]] := drive.motorAngVel;
	jointTorqueIn[phy2absMapping[driveIndex]] := drive.trqCalibrated;
	motorRefAnglesIn[phy2absMapping[driveIndex]] := drive.tgtAngle ;//当前参考角度，运动学输入
	
END_IF
END_METHOD

END_FUNCTION_BLOCK

// ---- POUs/tools/atan2Fun.TcPOU
FUNCTION atan2Fun : lreal
VAR_INPUT
	y:LREAL;
	x:LREAL;
END_VAR
VAR
END_VAR

//atan2(y,x)
IF ABS(x)<=0.0000001 THEN
	IF y>0 THEN
		atan2Fun:=pi/2;
	ELSE
		atan2Fun:=-pi/2;
	END_IF
ELSE
	IF x>0 THEN
		atan2Fun:=ATAN(y/x);
	ELSE
		IF y<0 THEN
			atan2Fun:=ATAN(y/x)-pi;	
		ELSE
			atan2Fun:=ATAN(y/x)+pi;
		END_IF
	END_IF
END_IF

END_FUNCTION

// ---- POUs/tools/CosGenerator.TcPOU
FUNCTION_BLOCK CosGenerator
VAR_INPUT
END_VAR
VAR_OUTPUT
	cosineSignalOut : LREAL;
END_VAR
VAR
	cosineSignal : LREAL;
	generatorCount : UDINT;
END_VAR

IF GVL.initCosGenerator THEN
	cosineSignal   := 0;   
	generatorCount := 0;
END_IF

IF GVL.cosStart THEN
   generatorCount := generatorCount + 1;
   cosineSignal := GVL.cosAmplitude * (1 - COS( 2 * pi * GVL.cosFrequency * generatorCount / 1.0 / gvl.sampleRate));
END_IF

IF GVL.cosStop THEN
   IF ABS(cosineSignal) < 0.00001 THEN  
	  GVL.cosStart  := FALSE;	
      GVL.cosStop   := FALSE;	
      generatorCount := 0;	  
   END_IF
END_IF

cosineSignalOut := cosineSignal;

END_FUNCTION_BLOCK

// ---- POUs/tools/VectorMath/SetMat7_3.TcPOU
FUNCTION SetMat7_3 :  ARRAY [0..6,0..2] OF int
VAR_INPUT
	x_11:INT;
	x_12:INT;
	x_13:INT;
	x_21:INT;
	x_22:INT;
	x_23:INT;
	x_31:INT;
	x_32:INT;
	x_33:INT;
	x_41:INT;
	x_42:INT;
	x_43:INT;
	x_51:INT;
	x_52:INT;
	x_53:INT;
	x_61:INT;
	x_62:INT;
	x_63:INT;
	x_71:INT;
	x_72:INT;
	x_73:INT;
END_VAR
VAR_OUTPUT
END_VAR
VAR
END_VAR

SetMat7_3 [0,0]:=x_11;
SetMat7_3 [0,1]:=x_12;
SetMat7_3 [0,2]:=x_13;

SetMat7_3 [1,0]:=x_21;
SetMat7_3 [1,1]:=x_22;
SetMat7_3 [1,2]:=x_23;

SetMat7_3 [2,0]:=x_31;
SetMat7_3 [2,1]:=x_32;
SetMat7_3 [2,2]:=x_33;

SetMat7_3 [3,0]:=x_41;
SetMat7_3 [3,1]:=x_42;
SetMat7_3 [3,2]:=x_43;

SetMat7_3 [4,0]:=x_51;
SetMat7_3 [4,1]:=x_52;
SetMat7_3 [4,2]:=x_53;

SetMat7_3 [5,0]:=x_61;
SetMat7_3 [5,1]:=x_62;
SetMat7_3 [5,2]:=x_63;

SetMat7_3 [6,0]:=x_71;
SetMat7_3 [6,1]:=x_72;
SetMat7_3 [6,2]:=x_73;

END_FUNCTION

// ---- POUs/tools/VectorMath/VecSum.TcPOU
FUNCTION VecSum : Vec3
VAR_INPUT
	a : ARRAY[0..3] OF Vec3; 
END_VAR
VAR
	i: INT;
	sum : Vec3;
END_VAR

sum := SetVec3(0, 0, 0);
FOR i := 0 TO 3 DO
	sum := VecAdd(sum, a[i]);
END_FOR
VecSum := sum;

END_FUNCTION

// ---- GlobalTextList.TcGTLO
TEXTLIST GlobalTextList
  20 = '%.2f'
  54 = '%.3f'
  66 = '%.4f'
  16 = '%d'
  11 = '%s'
  37 = 'AbsMove'
  23 = 'AbsStop'
  766 = 'ACE support'
  896 = 'Act Pos'
  136 = 'Act Trq'
  402 = 'Act Vel'
  10 = 'AddHeight'
  12 = 'AddHeightFrWalk'
  2481 = 'AddHFrWalk'
  1401 = 'adjust_angle (。)'
  1370 = 'adjust_angle（D）'
  1128 = 'adjust_angle（。）'
  408 = 'ALL'
  788 = 'All'
  779 = 'Arm'
  432 = 'ArmControl'
  578 = 'ArmRetract'
  1532 = 'ax'
  471 = 'Axis'
  184 = 'Axis Force Control'
  769 = 'Axis Group'
  750 = 'ay'
  1768 = 'az'
  613 = 'A_A'
  389 = 'A_S'
  636 = 'A_T'
  773 = 'BDF support'
  668 = 'BlegCenter'
  2058 = 'BLegPosAdjust'
  2185 = 'BLegRecovery'
  179 = 'BLegSlip control'
  1068 = 'Body phase'
  254 = 'BodyPosAdjust'
  453 = 'BPA ang (。)'
  905 = 'BPA x (m)'
  1485 = 'BPA y (m)'
  512 = 'B_A'
  539 = 'B_S'
  88 = 'B_T'
  626 = 'Cur Side Vel'
  993 = 'Cur Side Vel (A)'
  1378 = 'Cur Side Vel (B)'
  259 = 'Cur Trot Vel'
  575 = 'Cur Trot Vel (A)'
  931 = 'Cur Trot Vel (B)'
  522 = 'Cur Turn Vel'
  165 = 'Cur Turn Vel (A)'
  940 = 'Cur Turn Vel (B)'
  459 = 'Curling Control'
  1342 = 'Curling Control From Slip'
  84 = 'Curling Control From Stance'
  545 = 'CurlingFinished'
  710 = 'Current State'
  739 = 'C_A'
  206 = 'C_K'
  616 = 'C_S'
  880 = 'C_T'
  468 = 'Disable'
  388 = 'Drop'
  1095 = 'Drop height'
  564 = 'duration time'
  630 = 'Duty'
  868 = 'D_A'
  1288 = 'D_K'
  933 = 'D_S'
  34 = 'D_T'
  661 = 'Emergy STOP'
  69 = 'EN'
  1215 = 'Enable'
  797 = 'E_A'
  671 = 'E_S'
  576 = 'E_T'
  342 = 'FC'
  853 = 'fine adjust (。)'
  621 = 'FineTuning'
  1077 = 'FiveLegsLand'
  202 = 'FlegRotA'
  872 = 'FlegRotB'
  1014 = 'Force ctrl'
  120 = 'Force Ctrl Off'
  99 = 'Force Ctrl On'
  1183 = 'Force Stop'
  431 = 'Found'
  690 = 'FourLegsLand'
  100 = 'Foward Step length'
  140 = 'FRIC'
  343 = 'F_A'
  747 = 'F_S'
  195 = 'F_T'
  1569 = 'Gait Control'
  1512 = 'Hard'
  1337 = 'Height'
  70 = 'HM'
  644 = 'Home'
  902 = 'Impedance Control'
  855 = 'IMU'
  1231 = 'In BLeg Slip'
  573 = 'In TrotWalk'
  216 = 'increment_x'
  29 = 'increment_y'
  519 = 'increment_z'
  97 = 'Jog'
  385 = 'Jog Stop'
  113 = 'Jog Vel'
  1347 = 'Joint Ang'
  852 = 'Joint Trq'
  276 = 'KFI'
  1421 = 'KFP'
  1375 = 'KPD'
  186 = 'KPP'
  915 = 'Lateral Step length'
  796 = 'Leg A'
  1488 = 'Leg A adjInc'
  1199 = 'Leg A AdjInc'
  803 = 'Leg B'
  811 = 'Leg C'
  818 = 'Leg D'
  826 = 'Leg E'
  834 = 'Leg F'
  992 = 'Leg F AdjInc'
  1078 = 'Leg Status'
  412 = 'LegA'
  93 = 'LegA AdjInc'
  413 = 'LegB'
  414 = 'LegC'
  415 = 'LegD'
  416 = 'LegE'
  417 = 'LegF'
  1008 = 'LegF AdjInc'
  897 = 'LiftBody'
  999 = 'LiftMleg'
  349 = 'MlegRollA'
  96 = 'MlegRollB'
  743 = 'MlegRollC'
  268 = 'Motor Status'
  1259 = 'Move'
  1004 = 'OA ang (。)'
  67 = 'Op Mode'
  1419 = 'orient adjust (。)'
  393 = 'OrientAdjust'
  201 = 'P'
  1154 = 'Period'
  1239 = 'push vel (m/s)'
  28 = 'PushReleaseBall'
  1573 = 'Quit'
  1416 = 'R'
  168 = 'Rc control'
  1117 = 'Ready'
  223 = 'Recovery Curling'
  996 = 'ReduceHeight'
  1637 = 'ReduceHeightB'
  504 = 'ref ang initialization'
  1656 = 'Rep AC'
  1086 = 'Rep BLPA'
  825 = 'Rep BPA'
  378 = 'Rep OA'
  1420 = 'Rep RT'
  392 = 'Rep SP'
  226 = 'Rep SR'
  1372 = 'RepBC'
  838 = 'Req AC'
  379 = 'Req AH'
  874 = 'Req AHFW'
  148 = 'Req BC'
  988 = 'Req BLPA'
  1729 = 'Req BLR'
  265 = 'Req BPA'
  688 = 'Req CF'
  898 = 'Req FRA'
  712 = 'Req FRB'
  141 = 'Req FT'
  1219 = 'Req LML'
  857 = 'Req Move'
  737 = 'Req MRA'
  1241 = 'Req MRB'
  588 = 'Req MRC'
  1289 = 'Req OA'
  1114 = 'Req PRB'
  1911 = 'Req RC'
  1238 = 'Req RH'
  2068 = 'Req RHB'
  526 = 'Req RT'
  890 = 'Req SD'
  1162 = 'Req SL'
  638 = 'Req SP'
  719 = 'Req SR'
  783 = 'Req Stop'
  1406 = 'Req SU'
  801 = 'rough adjust (。)'
  1109 = 'RoughTuning'
  1990 = 'SearchPedal'
  1167 = 'Set colide'
  1649 = 'Set Impd'
  426 = 'Set Pos'
  475 = 'set ref angle'
  1157 = 'Set reference'
  409 = 'Shank'
  1217 = 'Short height'
  411 = 'Side'
  149 = 'Side Step'
  1038 = 'SixLegsLand'
  164 = 'Slide'
  1989 = 'slide Time(s)'
  1937 = 'Soft'
  1447 = 'Speed down Time(s)'
  390 = 'SpeedDown'
  1149 = 'SpeedUp'
  2211 = 'SraechPedal'
  552 = 'Start Gait'
  736 = 'Step ang'
  1483 = 'Step ang ((。)'
  547 = 'Step ang (。)'
  912 = 'Step Height'
  759 = 'Step height'
  27 = 'Step num'
  30 = 'StoneRot'
  1319 = 'stone_vel (RPM)'
  1218 = 'stone_vel(RPM)'
  92 = 'Stop'
  1424 = 'STOP'
  444 = 'Target Ang'
  1134 = 'target_vel (m/s)'
  1516 = 'target_vel(m/s)'
  865 = 'target_vel（m/s）'
  410 = 'Thigh'
  1063 = 'ThreeLegsLand'
  714 = 'Tip Actual Force     '
  257 = 'Tip Actual Position'
  787 = 'Tip Actual Velocity'
  188 = 'tip move'
  508 = 'Trgt Side Vel'
  705 = 'Trgt Trot Vel'
  530 = 'Trgt Turn Vel'
  713 = 'Trot control'
  176 = 'Trot Step'
  914 = 'Trq cmd'
  98 = 'Trq cmd (Emb)'
  1159 = 'Trq zero'
  772 = 'Turn Step'
  958 = 'Walk'
  672 = 'Y'
  549 = '休息'
  1471 = '侧移步长'
  65 = '停止'
  1788 = '前进步长'
  609 = '周期'
  1860 = '大腿抱角'
  2067 = '小腿抱角'
  2372 = '工作'
  394 = '摆动方向'
  55 = '斜坡行走'
  472 = '步高'
  467 = '滑行时间 (s)'
  1873 = '视觉运动(度)'
  311 = '转弯角度(度)'
  1082 = '降速时间(s)'
END_TEXTLIST

